TYPE "UDT_ModuleState"
TITLE = UDT_ModuleState
VERSION : 0.1
//User-defined structure of module states.
   STRUCT
      Configured { ExternalAccessible := 'False'; ExternalVisible := 'False'; ExternalWritable := 'False'} : Bool;   // Module configured
      Exist { ExternalAccessible := 'False'; ExternalVisible := 'False'; ExternalWritable := 'False'} : Bool;   // Module exist
      Error { ExternalAccessible := 'False'; ExternalVisible := 'False'; ExternalWritable := 'False'} : Bool;   // Module has error
   END_STRUCT;

END_TYPE

TYPE "UDT_DeviceState"
TITLE = UDT_DeviceState
VERSION : 0.1
//User-defined structure of device states.
   STRUCT
      Configure { ExternalAccessible := 'False'; ExternalVisible := 'False'; ExternalWritable := 'False'} : Bool;   // Device configured in TIA Portal hardware
      Exist { ExternalAccessible := 'False'; ExternalVisible := 'False'; ExternalWritable := 'False'} : Bool;   // Device physically connected
      Error { ExternalAccessible := 'False'; ExternalVisible := 'False'; ExternalWritable := 'False'} : Bool;   // Device has an error
      ProfinetNumber : UInt;   // Profinet slave number
      HW_ID : UInt;   // Device's HW_ID
      PNDeviceName : String;   // Device's project name
   END_STRUCT;

END_TYPE

TYPE "UDT_ProfinetDevice"
TITLE = UDT_ProfinetDevice
VERSION : 0.1
//User-defined structure of profinet device state.
   STRUCT
      DeviceState : "UDT_DeviceState";   // Device state
      Module { S7_SetPoint := 'False'} : Array[0..31] of "UDT_ModuleState";   // Modules
   END_STRUCT;

END_TYPE

TYPE "UDT_CommonStatus"
TITLE = UDT_CommonStatus
VERSION : 0.1
//User-defined structure of common statuses.
   STRUCT
      SafetyStop { ExternalAccessible := 'False'; ExternalVisible := 'False'; ExternalWritable := 'False'} : Bool;   // Emergancy stop
      Error { ExternalAccessible := 'False'; ExternalVisible := 'False'; ExternalWritable := 'False'} : Bool;   // An error is active
      Warning { ExternalAccessible := 'False'; ExternalVisible := 'False'; ExternalWritable := 'False'} : Bool;   // A warning is active
      ManualRun { ExternalAccessible := 'False'; ExternalVisible := 'False'; ExternalWritable := 'False'} : Bool;   // Running in manual mode
      Manual { ExternalAccessible := 'False'; ExternalVisible := 'False'; ExternalWritable := 'False'} : Bool;   // In manual mode
      Halted { ExternalAccessible := 'False'; ExternalVisible := 'False'; ExternalWritable := 'False'} : Bool;   // Halted
      Dieback { ExternalAccessible := 'False'; ExternalVisible := 'False'; ExternalWritable := 'False'} : Bool;   // In dieback
      Stopped { ExternalAccessible := 'False'; ExternalVisible := 'False'; ExternalWritable := 'False'} : Bool;   // Stopped
      Running { ExternalAccessible := 'False'; ExternalVisible := 'False'; ExternalWritable := 'False'} : Bool;   // Running
      EnergySave { ExternalAccessible := 'False'; ExternalVisible := 'False'; ExternalWritable := 'False'} : Bool;   // In energy saving mode
      AutoON { ExternalAccessible := 'False'; ExternalVisible := 'False'; ExternalWritable := 'False'} : Bool;   // Automatic started
   END_STRUCT;

END_TYPE

TYPE "UDT_ProfinetNetwork"
TITLE = UDT_ProfinetNetwork
VERSION : 0.1
//User-defined structure of profinet network state.
   STRUCT
      DeviceStatus : Array[0..512] of "UDT_ProfinetDevice";   // Profinet device status
   END_STRUCT;

END_TYPE

TYPE "UDT_GINWES"
VERSION : 0.1
   STRUCT
      Barcode : String[40];
   END_STRUCT;

END_TYPE

TYPE "UDT_GINWCS"
VERSION : 0.1
   STRUCT
      ActionTaken : String;   // Location code value that describes the actual disposition of the package
      Destination1 : String[20];   // Location code value that describes where the package should go (Diverter Number)
      Destination2 : String[20];   // Location code value that describes where the package should go (Diverter Number)
      Destination3 : String[20];   // Location code value that describes where the package should go (Diverter Number)
      Destination4 : String[20];   // Location code value that describes where the package should go (Diverter Number)
      Destination5 : String[20];   // Location code value that describes where the package should go (Diverter Number)
      ReasonCode : String[2];   // Management Code value that describes the result of attempting to route the package to the Destination
      Barcode1 : String;   // Barcode identifier code
      Barcode2 : String;
      Barcode3 : String;
      Barcode4 : String;
   END_STRUCT;

END_TYPE

TYPE "UDT_GINDHL"
VERSION : 0.1
   STRUCT
      ObjectID : String[10];   // Object ID
      VID : String[16];   // Virtual Item Identifier (VID)
      PieceID : String[40];   // Piece ID barcodes
      SortStrategy : String[1];   // Sort Strategy 1 - Highest priority available , 2 - Nearest
      ParcelReject { ExternalAccessible := 'False'; ExternalVisible := 'False'; ExternalWritable := 'False'} : Bool;   // True - Parcel reject
      Destination : Array[1..6] of Struct   // Destination
         ID : UInt;   // ID
         SortCommandActive { ExternalAccessible := 'False'; ExternalVisible := 'False'; ExternalWritable := 'False'} : Bool;   // Sort command
         ParcelSorted { ExternalAccessible := 'False'; ExternalVisible := 'False'; ExternalWritable := 'False'} : Bool;   // Parcel sorted
         Rejected { ExternalAccessible := 'False'; ExternalVisible := 'False'; ExternalWritable := 'False'} : Bool;   // Parcel rejected
         Reason : Int;   // Reason
      END_STRUCT;
      ParcelLocation : Struct   // Parcel Location
         Current : UInt;   // Current
         Last : UInt;   // Last
         Sort : UInt;   // Sort
      END_STRUCT;
      MFCMessage : Struct   // MFC Sort messages
         Sent : Struct   // Messages sent from the PLC to the MFC system
            SortResult { ExternalAccessible := 'False'; ExternalVisible := 'False'; ExternalWritable := 'False'} : Bool;   // Message Sort Result
            VIDResponse { ExternalAccessible := 'False'; ExternalVisible := 'False'; ExternalWritable := 'False'} : Bool;   // Message VID Response
            ScanReset { ExternalAccessible := 'False'; ExternalVisible := 'False'; ExternalWritable := 'False'} : Bool;   // Message Scan Reset
            XrayResult { ExternalAccessible := 'False'; ExternalVisible := 'False'; ExternalWritable := 'False'} : Bool;   // Message Xray result
            ParcelRegInfo { ExternalAccessible := 'False'; ExternalVisible := 'False'; ExternalWritable := 'False'} : Bool;   // Message Xray registration info
         END_STRUCT;
         Received : Struct   // Messages received from the MFC system to the PLC
            RejectParcel { ExternalAccessible := 'False'; ExternalVisible := 'False'; ExternalWritable := 'False'} : Bool;   // Message Reject Parcel
            Destination { ExternalAccessible := 'False'; ExternalVisible := 'False'; ExternalWritable := 'False'} : Bool;   // Message Destination
            DestinationResent { ExternalAccessible := 'False'; ExternalVisible := 'False'; ExternalWritable := 'False'} : Bool;   // Message Destination Resent
            TemporaryParcelIdentifier { ExternalAccessible := 'False'; ExternalVisible := 'False'; ExternalWritable := 'False'} : Bool;   // Message Temporary Parcel Identifier
            XrayRegistrationInfo { ExternalAccessible := 'False'; ExternalVisible := 'False'; ExternalWritable := 'False'} : Bool;
         END_STRUCT;
      END_STRUCT;
      Xray : Struct   // Xray data structure
         RoutingCode : String[2];   // Routing code
         Group : String[1];   // The group field is used to identify the group of the operator decisions came from in a
         Level : String[1];   // Level field is used to identify which level the operator decision came from in a
         Result : String[1];   // Results can be indicated with the following:A = Accept, R = Reject, U = Unavailable (Timeout), Z = High Threat
         BagIDMessage : Struct   // Message from PLC to Xray
            MessagePrepared { ExternalAccessible := 'False'; ExternalVisible := 'False'; ExternalWritable := 'False'} : Bool;   // The message is prepared and ready to send
            WrongMessageStructure { ExternalAccessible := 'False'; ExternalVisible := 'False'; ExternalWritable := 'False'} : Bool;   // The message has wrong structure
            Sent { ExternalAccessible := 'False'; ExternalVisible := 'False'; ExternalWritable := 'False'} : Bool;   // The message sent by PLC to Xray
            SentTime : String;   // Time when message sent by PLC to Xray
            NotSent { ExternalAccessible := 'False'; ExternalVisible := 'False'; ExternalWritable := 'False'} : Bool;   // The message was not sent from the PLC
            Received { ExternalAccessible := 'False'; ExternalVisible := 'False'; ExternalWritable := 'False'} : Bool;   // The message received by Xray
            TimeReceived : String;   // Time when message received by Xray
            NotReceived { ExternalAccessible := 'False'; ExternalVisible := 'False'; ExternalWritable := 'False'} : Bool;   // The message did not reach Xray
         END_STRUCT;
         DecisionMessage : Struct   // Message from Xray to PLC
            Received { ExternalAccessible := 'False'; ExternalVisible := 'False'; ExternalWritable := 'False'} : Bool;   // The message received by PLC
            ReceivedTime : String;   // The message received by PLC
            NotReceivedOnTime { ExternalAccessible := 'False'; ExternalVisible := 'False'; ExternalWritable := 'False'} : Bool;   // The message did not reach PLC
         END_STRUCT;
      END_STRUCT;
   END_STRUCT;

END_TYPE

TYPE "UDT_GINUPS"
VERSION : 0.1
   STRUCT
      TRKNUM : String[18];   // Tracking number
      PKGUID : String[32];   // Package ID
      MSGID : String[32];   // Message ID
      Length : Int;   // Camera Length in mm
      Width : Int;   // Camera Width in mm
      Height : Int;   // Camera Height in mm
      Weight : DInt;   // Weight in g
      IDCreated { ExternalAccessible := 'False'; ExternalVisible := 'False'; ExternalWritable := 'False'} : Bool;   // Byte 1, Bit 0 - PLCID created or TrayID Read
      DimDataRcv { ExternalAccessible := 'False'; ExternalVisible := 'False'; ExternalWritable := 'False'} : Bool;   // Byte 1, Bit 1 - Package Dimensional Data Received via Camera Scan Data Message
      PkgWrongInduct { ExternalAccessible := 'False'; ExternalVisible := 'False'; ExternalWritable := 'False'} : Bool;   // Byte 1, Bit 2 - Package Did NOT Induct Properly (Non-Tray Systems)
      IDCalcFromCamID { ExternalAccessible := 'False'; ExternalVisible := 'False'; ExternalWritable := 'False'} : Bool;   // Byte 2, Bit 0 - PLCID/TrayID Calculated From CamID
      UnknownParcelID { ExternalAccessible := 'False'; ExternalVisible := 'False'; ExternalWritable := 'False'} : Bool;   // Byte 2, Bit 4 - Unknown Parcel ID
      UndefinedProblem { ExternalAccessible := 'False'; ExternalVisible := 'False'; ExternalWritable := 'False'} : Bool;   // Byte 2, Bit 5 - Un-Defined Problem
      UnrecognizedCmd { ExternalAccessible := 'False'; ExternalVisible := 'False'; ExternalWritable := 'False'} : Bool;   // Byte 2, Bit 6 - Un-recognized command
      SorterInMainteneceMode { ExternalAccessible := 'False'; ExternalVisible := 'False'; ExternalWritable := 'False'} : Bool;   // Byte 2, Bit 7 - Sorter in Maintenance/Commissioning Mode
      DestUserSusp { ExternalAccessible := 'False'; ExternalVisible := 'False'; ExternalWritable := 'False'} : Bool;   // Byte 3, Bit 3 - Destination User Suspended
      SorterNotSynch { ExternalAccessible := 'False'; ExternalVisible := 'False'; ExternalWritable := 'False'} : Bool;   // Byte 3, Bit 6 - Sorter NOT Synchronized (Tilt Tray Systems)
      PkgDetAtVerCheckPoint { ExternalAccessible := 'False'; ExternalVisible := 'False'; ExternalWritable := 'False'} : Bool;   // Byte 4, Bit 0 - Package Detected at Verification Check Point
      ChuteFullAftrAlterDest { ExternalAccessible := 'False'; ExternalVisible := 'False'; ExternalWritable := 'False'} : Bool;   // Byte 4, Bit 7 - Preferred chute full after passed alternate destination
      ChuteNotAvailAfterAlterDest { ExternalAccessible := 'False'; ExternalVisible := 'False'; ExternalWritable := 'False'} : Bool;   // Byte 5, Bit 0 - Preferred chute not available after passed alternate destination
      PLCRedirected { ExternalAccessible := 'False'; ExternalVisible := 'False'; ExternalWritable := 'False'} : Bool;   // Byte 5, Bit 2 - PLC Redirected
      ThreatParcel { ExternalAccessible := 'False'; ExternalVisible := 'False'; ExternalWritable := 'False'} : Bool;   // Threat parcel
   END_STRUCT;

END_TYPE

TYPE "UDT_GINFedEx"
VERSION : 0.1
   STRUCT
      Timestamp : String[17];   // Local time timestamp
      TimeZoneDesignator : String[5];   // Time zone designator
      PackageEntrancePoint : String[14];   // Entrance point, where LLC starts tracking the parcel.
      PackageEntranceState : String[1];   // Entrance state
      PackageExitPoint : String[14];   // Exit point name, where LLC reports the last known tracking point.
      PackageExitState : String[1];   // Exit point state when LLC reports the last known tracking point.
      PalletType : String[2];   // Pallet code for different type of pallets on the market
      Mask : String[1];   // Flag to indicate that a pallet has been mask.
      CellNumber : String[4];   // Tray/Cell number (for loop sorters) or generated by LLC (on line sorters).
      CellsOccupied : String[1];   // Cells occupied by the piece for loop sorters.
      ImageID : String[6];   // Image ID number created by the ADC system.
      ScanUnitType : String[1];   // Scan unit type
      ADCSystemID : String[15];   // Number assigned by the ADC system
      PackageID : String[15];   // Number assigned by the LLC system
      LLCSystemID : String[15];
      HLCPackageID : String[10];   // Unique number for the specific package during it stays in HLC system.
      HLCResultCode : String[16];   // Result code based on processing of the scan event messages.
      ShipmentID : String[6];   // Consignment id of the parcel.
      WeightStatus : String[1];   // Status to indicate if the parcel/pallet has weight on the system.
      ActualDestination : String[6];   // Location code value that describes the actual disposition of the package.
      Destination1 : String[6];   // Location code value that describes where the package should go (Diverter Number).
      Destination2 : String[6];   // Location code value that describes where the package should go (Diverter Number).
      Destination3 : String[6];   // Location code value that describes where the package should go (Diverter Number).
      Destination4 : String[6];   // Location code value that describes where the package should go (Diverter Number).
      Destination5 : String[6];   // Location code value that describes where the package should go (Diverter Number).
      CutOffTimeDestination1 : String[5];   // Cut Off Time in Local Time.
      CutOffTimeDestination2 : String[5];   // Cut Off Time in Local Time.
      CutOffTimeDestination3 : String[5];   // Cut Off Time in Local Time.
      CutOffTimeDestination4 : String[5];   // Cut Off Time in Local Time.
      CutOffTimeDestination5 : String[5];   // Cut Off Time in Local Time.
      ReasonCode1 : String[8];   // Management Code value that describes the result of attempting to route the package to the Destination
      ReasonCode2 : String[8];   // Management Code value that describes the result of attempting to route the package to the Destination
      ReasonCode3 : String[8];   // Management Code value that describes the result of attempting to route the package to the Destination
      ReasonCode4 : String[8];   // Management Code value that describes the result of attempting to route the package to the Destination
      ReasonCode5 : String[8];   // Management Code value that describes the result of attempting to route the package to the Destination
      HLCDataText : String[20];   // Free text for future use.
      Customs : String[1];   // Need to be checked by customs
      DIMSystemID : String[15];   // Identifier of dimensioning system.
      DIMStatus : String[5];   // Basic diagnostic information from the dimensioning system at the moment of the measurement.
      PackageDimLength : String[6];   // Length dimension of package in resolution of dim system.
      PackageDimWidth : String[6];   // Width dimension of package in resolution of dim system.
      PackageDimHeight : String[6];   // Height dimension of package in resolution of dim system.
      DIMUOM : String[2];   // Unit of measure of the package dimensions.
      DimLFTstatusCode : String[8];   // Dimension LFT status code.
      DimConfidence : String[2];   // The level of assurance for the correct dimensions.
      DimensionSource : String[1];   // For combined camera/laser dim acquisition devices. It indicates type of capturing mode
      AlibiDims : String[25];   // Alibi for Dimensions
      SCLSystemID : String[15];   // Identifier of weight scale.
      SCLStatus : String[5];   // Basic diagnostic information from the weight scale system.
      SCLWT : String[6];   // Scale weight of package in resolution of scale system.
      SCLWTUOM : String[2];   // Unit of measurement for Weight
      SCLLFTStatusCode : String[2];   // Scale LFT status code.
      AlibiWeight : String[25];   // Alibi for Weight
      ReasonCode : String[1];   // This code should be used when the SI message has some defect.
      Stackable : String[1];   // If stackable recognition is enabled, Y or N
      Stickerstype : String[2];   // When optical recognition is used to sort
      FlyingDocument : String[1];   // Status to confirm if the document/flyer is prone to fly off the sorter.
      ModeofOperation : String[1];   // Camera Tunnel operational mode format:
      CameraHeadstatus : String[2];   // Diagnostic information on camera/laser heads performing barcode reads.
      PackageDataTruncated : String[1];   // Y = Full length of barcode data exceeds 9999 bytes, data truncated
      TotalBarcodeDataLength : String[4];   // Length of all barcode data that was sent in bytes;
      Barcode1Identification : String[3];   // Barcode identifier code.
      Barcode1status : String[2];   // Barcode confidence factor
      Barcode1datalength : String[4];   // String length of barcode data in bytes; inclusive of this field. Use 0054 as a fixed value
      Barcode1data : String[50];   // Highest priority barcode
      Barcode2Identification : String[3];   // Barcode identifier code.
      Barcode2status : String[2];   // Barcode confidence factor
      Barcode2datalength : String[4];   // String length of barcode data in bytes; inclusive of this field. Use 0054 as a fixed value
      Barcode2data : String[50];   // Highest priority barcode
      Barcode3Identification : String[3];   // Barcode identifier code.
      Barcode3status : String[2];   // Barcode confidence factor
      Barcode3datalength : String[4];   // String length of barcode data in bytes; inclusive of this field. Use 0054 as a fixed value
      Barcode3data : String[50];   // Highest priority barcode
      BarcodeIdentification : String[3];   // Barcode identifier code.
      Barcodestatus : String[2];   // Barcode confidence factor
      Barcodedatalength : String[4];   // String length of barcode data in bytes
      Barcodedata : String[50];   // Sortation barcode
      CustomerID : DInt;   // 6 digits SequentialID (NNNNNN)
      AreaNumber : String[2];   // Package Sequence ID "Area Number"
      PurgeEnabled { ExternalAccessible := 'False'; ExternalVisible := 'False'; ExternalWritable := 'False'} : Bool;   // Purge enabled for parcel: destination overwritten with Purge destination
   END_STRUCT;

END_TYPE

TYPE "UDT_GINStandard"
VERSION : 0.1
   STRUCT
      Destination : Array[0..20] of DInt;   // Destination
      Identification : Struct   // Barcode identification
         GoodRead { ExternalAccessible := 'False'; ExternalVisible := 'False'; ExternalWritable := 'False'} : Bool;   // Barcode read was succesful
         NoRead { ExternalAccessible := 'False'; ExternalVisible := 'False'; ExternalWritable := 'False'} : Bool;   // Barcode read was unsuccesful
         MultiRead { ExternalAccessible := 'False'; ExternalVisible := 'False'; ExternalWritable := 'False'} : Bool;   // Multiple Barcodes were detected
         Barcode : Array[0..10] of Char;   // Barcode values
      END_STRUCT;
      GinAssigned { ExternalAccessible := 'False'; ExternalVisible := 'False'; ExternalWritable := 'False'} : Bool;   // GIN is assigned to package
      Lost { ExternalAccessible := 'False'; ExternalVisible := 'False'; ExternalWritable := 'False'} : Bool;   // Lost in tracking
      Length : Int;   // Length in mm
      Width : Int;   // Width in mm
      Height : Int;   // Height in mm
      Weight : DInt;   // Weight in g
      PkgTooLong { ExternalAccessible := 'False'; ExternalVisible := 'False'; ExternalWritable := 'False'} : Bool;   // Package is too long
      PkgTooSmall { ExternalAccessible := 'False'; ExternalVisible := 'False'; ExternalWritable := 'False'} : Bool;   // Package is too small
      PkgTooHigh { ExternalAccessible := 'False'; ExternalVisible := 'False'; ExternalWritable := 'False'} : Bool;   // Package is too high
      PkgOverWeight { ExternalAccessible := 'False'; ExternalVisible := 'False'; ExternalWritable := 'False'} : Bool;   // Package is over weight
      TrailingGap : Int;   // Trailing gap size in cm between the package
      LeadingGap : Int;   // Leading gap size in cm between the package
      NrOfRecirculations : Int;   // Number of recirculations
      DestReqSend { ExternalAccessible := 'False'; ExternalVisible := 'False'; ExternalWritable := 'False'} : Bool;   // Destination request sent to high level
      DestRcv { ExternalAccessible := 'False'; ExternalVisible := 'False'; ExternalWritable := 'False'} : Bool;   // Destination received from high level
      SortStatus : Struct   // Sort status of the package
         DivertDestination : Int;   // Destination to which the package is diverted
         GoodDivert { ExternalAccessible := 'False'; ExternalVisible := 'False'; ExternalWritable := 'False'} : Bool;   // Package diverted
         FailedDivert { ExternalAccessible := 'False'; ExternalVisible := 'False'; ExternalWritable := 'False'} : Bool;   // Package failed to divert
         NoDivert : Bool := TRUE;   // Divert is not activated
         NoDivertCause : Struct   // Cause for no divert
            ChuteJam { ExternalAccessible := 'False'; ExternalVisible := 'False'; ExternalWritable := 'False'} : Bool;   // Chute is jammed
            ChuteFull { ExternalAccessible := 'False'; ExternalVisible := 'False'; ExternalWritable := 'False'} : Bool;   // Chute is full
            NoRTR { ExternalAccessible := 'False'; ExternalVisible := 'False'; ExternalWritable := 'False'} : Bool;   // Downstream conveyor is not ready to receive
            DestDisabled { ExternalAccessible := 'False'; ExternalVisible := 'False'; ExternalWritable := 'False'} : Bool;   // Destination is disabled
            TrayDisabled { ExternalAccessible := 'False'; ExternalVisible := 'False'; ExternalWritable := 'False'} : Bool;   // Tray is disabled
            SorterNotAtSpeed { ExternalAccessible := 'False'; ExternalVisible := 'False'; ExternalWritable := 'False'} : Bool;   // Sorter is not at speed
            LeadingGapError { ExternalAccessible := 'False'; ExternalVisible := 'False'; ExternalWritable := 'False'} : Bool;   // Gap size with downstream parcel is not enough
            TrailingGapError { ExternalAccessible := 'False'; ExternalVisible := 'False'; ExternalWritable := 'False'} : Bool;   // Gap size with upstream parcel is not enough
            PkgTooHigh { ExternalAccessible := 'False'; ExternalVisible := 'False'; ExternalWritable := 'False'} : Bool;   // Package is too high to divert
            PkgTooLong { ExternalAccessible := 'False'; ExternalVisible := 'False'; ExternalWritable := 'False'} : Bool;   // Package is too long to divert
            DestNotReachable { ExternalAccessible := 'False'; ExternalVisible := 'False'; ExternalWritable := 'False'} : Bool;   // Sort destionation is not reachable
            InvalidDest { ExternalAccessible := 'False'; ExternalVisible := 'False'; ExternalWritable := 'False'} : Bool;   // Sort destination is invalid
            DestTooLate { ExternalAccessible := 'False'; ExternalVisible := 'False'; ExternalWritable := 'False'} : Bool;   // Destination too late
            NoDestRcv { ExternalAccessible := 'False'; ExternalVisible := 'False'; ExternalWritable := 'False'} : Bool;   // Destination not received from high level
         END_STRUCT;
      END_STRUCT;
   END_STRUCT;

END_TYPE

TYPE "UDT_EventStatistic"
TITLE = UDT_EventStatistic
VERSION : 0.1
//User-defined structure of event statistic data.
   STRUCT
      NumberOfTimes : DInt;   // Number of times the event occurred since last reset
      LastEventSeconds : DInt;   // Number of seconds of the current or last event
      TotalEventSeconds : DInt;   // Total number of seconds the event occurred since last reset
   END_STRUCT;

END_TYPE

FUNCTION "FC_GetNrOfArrayEl" : Int
TITLE = FC_GetNrOfArrayEl
{ S7_Optimized_Access := 'TRUE' }
AUTHOR : MHSE
FAMILY : GeneralSystemFunctions
VERSION : 3.0
// ATTRIBUTES
// AUTO_NUMBER = True
// BLOCK_NUMBER = 19
// END_ATTRIBUTES
//Function to get the number of array elements.
   VAR_INPUT
      iv_Array : Variant;   // Input array
   END_VAR

   VAR_TEMP
      ti_NrOfArrayEl : Int;   // Number of array elements
   END_VAR


BEGIN
	(*
	----------------------------------------------------------------------------------------

	Version history:
	Date        | Version   | Author        | Remark
	----------------------------------------------------------------------------------------
	24/05/2019  | 0.1       | L.Klar        | first release MHS TIA 15.1
	24/07/2019  | 2.0       | L.Klar        | 2.0 MHS library release TIA 15.1
	27/08/2019  | 2.1       | K.Pokorski    | Comments adjusted
	12/11/2019  | 3.0       | P.Majka       | 3.0 MHS library release TIA 15.1
	21/02/2023  | 4.0       | F.Baten       | 4.0 Release TIA 17.5
	*)

	REGION 1 – Number of an array elements

	    IF IS_ARRAY(#iv_Array)                                                  // Input variable is an array
	    THEN

	        #ti_NrOfArrayEl := UDINT_TO_INT(CountOfElements(#iv_Array));

	        // Reset array length if the input variable isn't an array
	    ELSE

	        #ti_NrOfArrayEl := 0;

	    END_IF;

	END_REGION

	REGION 2 – Return output

	    #FC_GetNrOfArrayEl := #ti_NrOfArrayEl;

	END_REGION

END_FUNCTION

TYPE "UDT_AixMotorStatus"
VERSION : 0.1
   STRUCT
      Overheat { ExternalAccessible := 'False'; ExternalVisible := 'False'; ExternalWritable := 'False'} : Bool;   // Motor temperature has exceeded 105 degrees Celsius
      MaxTorque { ExternalAccessible := 'False'; ExternalVisible := 'False'; ExternalWritable := 'False'} : Bool;   // Motor at maximum torque output
      ShortCircuit { ExternalAccessible := 'False'; ExternalVisible := 'False'; ExternalWritable := 'False'} : Bool;   // Motor short circuit
      MotorNotConnected { ExternalAccessible := 'False'; ExternalVisible := 'False'; ExternalWritable := 'False'} : Bool;   // Motor is not connected
      Overload { ExternalAccessible := 'False'; ExternalVisible := 'False'; ExternalWritable := 'False'} : Bool;   // Motor overloaded after more than 20 seconds in Stalled
      Stalled { ExternalAccessible := 'False'; ExternalVisible := 'False'; ExternalWritable := 'False'} : Bool;   // Motor stalled and speed is less than 10% of the set speed
      BadHall { ExternalAccessible := 'False'; ExternalVisible := 'False'; ExternalWritable := 'False'} : Bool;   // Motor Hall Effect Sensor error active
      MotorNotUsed { ExternalAccessible := 'False'; ExternalVisible := 'False'; ExternalWritable := 'False'} : Bool;   // Motor is not used
      MotorStatus1 { ExternalAccessible := 'False'; ExternalVisible := 'False'; ExternalWritable := 'False'} : Bool;   // Motor running and direction status
      MotorStatus2 { ExternalAccessible := 'False'; ExternalVisible := 'False'; ExternalWritable := 'False'} : Bool;   // Motor running and direction status
      MotorPortinDOmode { ExternalAccessible := 'False'; ExternalVisible := 'False'; ExternalWritable := 'False'} : Bool;   // Motor port is in digital output mode .
      Bit03 { ExternalAccessible := 'False'; ExternalVisible := 'False'; ExternalWritable := 'False'} : Bool;   // Reserved
      Bit04 { ExternalAccessible := 'False'; ExternalVisible := 'False'; ExternalWritable := 'False'} : Bool;   // Reserved
      BoardOverheat { ExternalAccessible := 'False'; ExternalVisible := 'False'; ExternalWritable := 'False'} : Bool;   // Reserved
      OverVoltage { ExternalAccessible := 'False'; ExternalVisible := 'False'; ExternalWritable := 'False'} : Bool;   // Supply voltage + motor back EMF exceeded 30 volts
      LowVoltage { ExternalAccessible := 'False'; ExternalVisible := 'False'; ExternalWritable := 'False'} : Bool;   // Module power supply is less than 18 Volts
      MotorStatus : DWord;
   END_STRUCT;

END_TYPE

TYPE "UDT_EquipmentControl"
TITLE = UDT_EquipmentControl
VERSION : 0.1
//User-defined structure of equipment control commands.
   STRUCT
      Command : Struct   // Control command
         Start { ExternalAccessible := 'False'; ExternalVisible := 'False'; ExternalWritable := 'False'} : Bool;   // Start conveyor
         Stop { ExternalAccessible := 'False'; ExternalVisible := 'False'; ExternalWritable := 'False'} : Bool;   // Stop conveyor
         Reset { ExternalAccessible := 'False'; ExternalVisible := 'False'; ExternalWritable := 'False'} : Bool;   // Faults reset
         ResetData { ExternalAccessible := 'False'; ExternalVisible := 'False'; ExternalWritable := 'False'} : Bool;   // Statistics reset
         ManualMode { ExternalAccessible := 'False'; ExternalVisible := 'False'; ExternalWritable := 'False'} : Bool;   // Manual mode required
         DisableManualMode { ExternalAccessible := 'False'; ExternalVisible := 'False'; ExternalWritable := 'False'} : Bool;   // Disable manual mode
         AutomaticOn { ExternalAccessible := 'False'; ExternalVisible := 'False'; ExternalWritable := 'False'} : Bool;   // System is started in automatic mode
         StopRequest { ExternalAccessible := 'False'; ExternalVisible := 'False'; ExternalWritable := 'False'} : Bool;
      END_STRUCT;
      Report { S7_SetPoint := 'False'} : "UDT_CommonStatus";   // Conveyors state
      Request : Struct   // Request from equipment
         RestartRequired { ExternalAccessible := 'False'; ExternalVisible := 'False'; ExternalWritable := 'False'} : Bool;   // Restart required from system control
         SignalingRequest { ExternalAccessible := 'False'; ExternalVisible := 'False'; ExternalWritable := 'False'} : Bool;   // Beeper required
         InhibitStop { ExternalAccessible := 'False'; ExternalVisible := 'False'; ExternalWritable := 'False'} : Bool;
      END_STRUCT;
   END_STRUCT;

END_TYPE

DATA_BLOCK "DB_ProfinetDiagnostic"
TITLE = DB_ProfinetDiagnostic
{ S7_Optimized_Access := 'TRUE' }
AUTHOR : MHSE
FAMILY : GeneralSystemFunctions
VERSION : 3.0
NON_RETAIN
//Data block to store profinet network diagnostic data.
   VAR
      ProfinetNetworks { ExternalAccessible := 'False'; ExternalVisible := 'False'; ExternalWritable := 'False'; S7_SetPoint := 'False'} : Array[1..10] of "UDT_ProfinetNetwork";
   END_VAR


BEGIN

END_DATA_BLOCK

TYPE "UDT_GIN"
VERSION : 0.1
   STRUCT
      General { S7_SetPoint := 'False'} : "UDT_GINStandard";
      FedEx { S7_SetPoint := 'False'} : "UDT_GINFedEx";
      UPS { S7_SetPoint := 'False'} : "UDT_GINUPS";
      DHL { S7_SetPoint := 'False'} : "UDT_GINDHL";
      WCS { S7_SetPoint := 'False'} : "UDT_GINWCS";
      WES { S7_SetPoint := 'False'} : "UDT_GINWES";
   END_STRUCT;

END_TYPE

DATA_BLOCK "DB_Memory"
TITLE = DB_Memory
{ S7_Optimized_Access := 'TRUE' }
AUTHOR : MHSE
VERSION : 3.0
NON_RETAIN
   VAR
      ClockByte { ExternalAccessible := 'False'; ExternalVisible := 'False'; ExternalWritable := 'False'} : Byte;   // System clock byte
      Clock_10Hz { ExternalAccessible := 'False'; ExternalVisible := 'False'; ExternalWritable := 'False'} : Bool;   // 10 Hz system clock bit
      Clock_5Hz { ExternalAccessible := 'False'; ExternalVisible := 'False'; ExternalWritable := 'False'} : Bool;   // 5 Hz system clock bit
      "Clock_2.5Hz" { ExternalAccessible := 'False'; ExternalVisible := 'False'; ExternalWritable := 'False'} : Bool;   // 2.5 Hz system clock bit
      Clock_2Hz { ExternalAccessible := 'False'; ExternalVisible := 'False'; ExternalWritable := 'False'} : Bool;   // 2 Hz system clock bit
      "Clock_1.25Hz" { ExternalAccessible := 'False'; ExternalVisible := 'False'; ExternalWritable := 'False'} : Bool;   // 1.25 Hz system clock bit
      Clock_1Hz { ExternalAccessible := 'False'; ExternalVisible := 'False'; ExternalWritable := 'False'} : Bool;   // 1 Hz system clock bit
      "Clock_0.625Hz" { ExternalAccessible := 'False'; ExternalVisible := 'False'; ExternalWritable := 'False'} : Bool;   // 0.625 Hz system clock bit
      "Clock_0.5Hz" { ExternalAccessible := 'False'; ExternalVisible := 'False'; ExternalWritable := 'False'} : Bool;   // 0.5 Hz system clock bit
      SystemByte { ExternalAccessible := 'False'; ExternalVisible := 'False'; ExternalWritable := 'False'} : Byte;   // System byte
      OSClockByte { ExternalAccessible := 'False'; ExternalVisible := 'False'; ExternalWritable := 'False'} : Byte;   // One shot of clock pulse
      "OS_0.1sec" { ExternalAccessible := 'False'; ExternalVisible := 'False'; ExternalWritable := 'False'} : Bool;   // One shot every 0.1 sec
      "OS_0.2sec" { ExternalAccessible := 'False'; ExternalVisible := 'False'; ExternalWritable := 'False'} : Bool;   // One shot every 0.2 sec
      "OS_0.4sec" { ExternalAccessible := 'False'; ExternalVisible := 'False'; ExternalWritable := 'False'} : Bool;   // One shot every 0.4 sec
      "OS_0.5sec" { ExternalAccessible := 'False'; ExternalVisible := 'False'; ExternalWritable := 'False'} : Bool;   // One shot every 0.5 sec
      "OS_0.8sec" { ExternalAccessible := 'False'; ExternalVisible := 'False'; ExternalWritable := 'False'} : Bool;   // One shot every 0.8 sec
      OS_1sec { ExternalAccessible := 'False'; ExternalVisible := 'False'; ExternalWritable := 'False'} : Bool;   // One shot every 1 sec
      "OS_1.6sec" { ExternalAccessible := 'False'; ExternalVisible := 'False'; ExternalWritable := 'False'} : Bool;   // One shot every 1.6 sec
      OS_2sec { ExternalAccessible := 'False'; ExternalVisible := 'False'; ExternalWritable := 'False'} : Bool;   // One shot every 2 sec
      PrevCycleTime { ExternalAccessible := 'False'; ExternalVisible := 'False'; ExternalWritable := 'False'} : LReal;   // Previous PLC cycle Time
      RuntimeMem { ExternalAccessible := 'False'; ExternalVisible := 'False'; ExternalWritable := 'False'} : LReal;   // Runtime memory
      FirstScan { ExternalAccessible := 'False'; ExternalVisible := 'False'; ExternalWritable := 'False'} : Bool;   // First scan bit
      DiagStatusUpdate { ExternalAccessible := 'False'; ExternalVisible := 'False'; ExternalWritable := 'False'} : Bool;   // Diagnostic status update
      AlwaysTrue { ExternalAccessible := 'False'; ExternalVisible := 'False'; ExternalWritable := 'False'} : Bool;   // Always True bit
      AlwaysFalse { ExternalAccessible := 'False'; ExternalVisible := 'False'; ExternalWritable := 'False'} : Bool;   // Always False bit
      CommissioningFalse { ExternalAccessible := 'False'; ExternalVisible := 'False'; ExternalWritable := 'False'} : Bool;   // Commissioning always false
      CommissioningTrue { ExternalAccessible := 'False'; ExternalVisible := 'False'; ExternalWritable := 'False'} : Bool;   // Commissioning always true
      ReconnectCommand { ExternalAccessible := 'False'; ExternalVisible := 'False'; ExternalWritable := 'False'} : Bool;   // Reconnect command
      ScanMainRack { ExternalAccessible := 'False'; ExternalVisible := 'False'; ExternalWritable := 'False'} : Bool;   // Trigger to check main rack confiuration
      ScanProfinet { ExternalAccessible := 'False'; ExternalVisible := 'False'; ExternalWritable := 'False'} : Bool;   // Scan profinet bit
      Simulation { ExternalAccessible := 'False'; ExternalVisible := 'False'; ExternalWritable := 'False'} : Bool;   // Simulation
      PN1OK { ExternalAccessible := 'False'; ExternalVisible := 'False'; ExternalWritable := 'False'} : Bool;   // Profinet ok
      "Local~PROFINET_IO-System" { ExternalAccessible := 'False'; ExternalVisible := 'False'; ExternalWritable := 'False'} : HW_ANY;   // HW Intentifier of PN-IO System
      "Local~PROFINET_IO-System_1" { ExternalAccessible := 'False'; ExternalVisible := 'False'; ExternalWritable := 'False'} : HW_ANY;   // HW Intentifier of PN-IOSystem 1
      "Local~PROFINET_IO-System_2" { ExternalAccessible := 'False'; ExternalVisible := 'False'; ExternalWritable := 'False'} : HW_ANY;   // HW Intentifier of PN-IOSystem 2
      "Local~PROFINET_IO-System_3" { ExternalAccessible := 'False'; ExternalVisible := 'False'; ExternalWritable := 'False'} : HW_ANY;   // HW Intentifier of PN-IOSystem 3
      "Local~PROFINET_IO-System_4" { ExternalAccessible := 'False'; ExternalVisible := 'False'; ExternalWritable := 'False'} : HW_ANY;   // HW Intentifier of PN-IOSystem 4
      "Local~PROFINET_IO-System_5" { ExternalAccessible := 'False'; ExternalVisible := 'False'; ExternalWritable := 'False'} : HW_ANY;   // HW Intentifier of PN-IOSystem 5
      "Local~PROFINET_IO-System_6" { ExternalAccessible := 'False'; ExternalVisible := 'False'; ExternalWritable := 'False'} : HW_ANY;   // HW Intentifier of PN-IOSystem 6
      "Local~PROFINET_IO-System_7" { ExternalAccessible := 'False'; ExternalVisible := 'False'; ExternalWritable := 'False'} : HW_ANY;   // HW Intentifier of PN-IOSystem 7
      "Local~PROFINET_IO-System_8" { ExternalAccessible := 'False'; ExternalVisible := 'False'; ExternalWritable := 'False'} : HW_ANY;   // HW Intentifier of PN-IOSystem 8
      "Local~PROFINET_IO-System_9" { ExternalAccessible := 'False'; ExternalVisible := 'False'; ExternalWritable := 'False'} : HW_ANY;   // HW Intentifier of PN-IOSystem 9
   END_VAR


BEGIN

END_DATA_BLOCK

TYPE "UDT_PNDevice"
VERSION : 0.1
   STRUCT
      PNNetworknumber : Int := 1;   // Number of the profinet network where device exist
      PNDeviceNumber : Int := 0;   // Profinet number of the device
      PNDeviceFound { ExternalAccessible := 'False'; ExternalVisible := 'False'; ExternalWritable := 'False'} : Bool;   // Device found in Profinet structure
   END_STRUCT;

END_TYPE

TYPE "UDT_VfdSinaParameterUser"
TITLE = UDT_VFD_SinaParameterUser
VERSION : 0.1
//User-defined structure of Siemens parameter.
   STRUCT
      siParaNo : UInt;   // Number of parameter (Number 1..65535)
      siIndex : Int;   // Subindex (Number 1..65535)
      srValue : Real;   // Value of parameter
      sdValue : DInt;   // Value of parameter
      syFormat : Byte := BYTE#16#00;   // Format of value (Format 0x40..0x44)
      swErrorNo : Word := WORD#16#0000;   // Error number (see table below)
   END_STRUCT;

END_TYPE

TYPE "UDT_ConveyorCommonConfiguration"
VERSION : 0.1
   STRUCT
      Length : DInt;   // Conveyor length [mm]
      LengthCorrection : DInt;   // Length correction [mm]
   END_STRUCT;

END_TYPE

TYPE "UDT_InductParcelData"
VERSION : 0.1
   STRUCT
      GINNumber : Int;   // GIN number
      GapRequired : Int;   // Size of gap requested by induct
      WindowPosition : Int;   // Position of the window in the merge tracking
      WindowReserved { ExternalAccessible := 'False'; ExternalVisible := 'False'; ExternalWritable := 'False'} : Bool;   // The window is reserved for the induct
   END_STRUCT;

END_TYPE

FUNCTION_BLOCK "FB_OnOffDelayDistance"
TITLE = FB_TimerOnOffDelay
{ S7_Optimized_Access := 'TRUE' }
AUTHOR : MHSE
FAMILY : GeneralSystemFunctions
VERSION : 3.0
// ATTRIBUTES
// AUTO_NUMBER = True
// BLOCK_NUMBER = 18
// END_ATTRIBUTES
//Function block to generate on/off signal delay.
   VAR_INPUT
      idi_OnDelayDistance { ExternalAccessible := 'False'; ExternalVisible := 'False'; ExternalWritable := 'False'} : DInt;   // On delay distance [cm]
      idi_OffDelayDistance { ExternalAccessible := 'False'; ExternalVisible := 'False'; ExternalWritable := 'False'} : DInt;   // Off delay distance [cm]
      ii_Displacement { ExternalAccessible := 'False'; ExternalVisible := 'False'; ExternalWritable := 'False'} : Int;   // Actual displacement
      ix_SignalToDelay { ExternalAccessible := 'False'; ExternalVisible := 'False'; ExternalWritable := 'False'} : Bool;   // Input signal to be delayed
      ix_Enable { ExternalAccessible := 'False'; ExternalVisible := 'False'; ExternalWritable := 'False'} : Bool := TRUE;   // Measuring enable
   END_VAR

   VAR_OUTPUT
      qdi_ActualDelayDistance { ExternalAccessible := 'False'; ExternalVisible := 'False'; ExternalWritable := 'False'} : DInt;   // Actual delay distance [cm]
      qx_DelayedSignal { ExternalAccessible := 'False'; ExternalVisible := 'False'; ExternalWritable := 'False'} : Bool;   // Delayed signal output
   END_VAR

   VAR RETAIN
      sdi_ActualDelayDistance { ExternalAccessible := 'False'; ExternalVisible := 'False'; ExternalWritable := 'False'} : DInt;   // Actual delay distance [cm]
   END_VAR
   VAR
      s_R_TRIG_Signal {InstructionName := 'R_TRIG'; LibVersion := '1.0'; ExternalAccessible := 'False'; ExternalVisible := 'False'; ExternalWritable := 'False'; S7_SetPoint := 'False'} : R_TRIG;   // Siemens "R_Trig" - to prepare the rising edge trigger on "ix_SignalToDelay" signal
      s_F_TRIG_Signal {InstructionName := 'F_TRIG'; LibVersion := '1.0'; ExternalAccessible := 'False'; ExternalVisible := 'False'; ExternalWritable := 'False'; S7_SetPoint := 'False'} : F_TRIG;   // Siemens "F_Trig" - to prepare the falling edge trigger on "ix_SignalToDelay" signal
   END_VAR


BEGIN
	(*
	----------------------------------------------------------------------------------------

	Version history:
	Date        | Version   | Author        | Remark
	----------------------------------------------------------------------------------------
	26/04/2023  | 0.1       | F.Baten       | first release MHS TIA 15.1
	*)

	REGION Step 1 – Input signal edge detection

	    #s_R_TRIG_Signal(CLK := #ix_SignalToDelay);


	    #s_F_TRIG_Signal(CLK := #ix_SignalToDelay);

	END_REGION

	REGION Step 2 – Actual delay distance initialization

	    IF (#s_R_TRIG_Signal.Q OR #s_F_TRIG_Signal.Q)           // Input signal changed
	    THEN

	        #sdi_ActualDelayDistance := 0;

	    END_IF;

	END_REGION

	REGION Step 3 – On/Off delay distance calculation


	    IF (#ix_SignalToDelay                                       // Signal to be delayed is active
	        AND #ix_Enable)                                         // Measuring enabled
	    THEN

	        // Timer on
	        IF (#sdi_ActualDelayDistance >= #idi_OnDelayDistance)
	        THEN

	            #qx_DelayedSignal := TRUE;

	        ELSE

	            #sdi_ActualDelayDistance += ABS(#ii_Displacement);

	        END_IF;

	    END_IF;

	    // Timer off
	    IF (NOT #ix_SignalToDelay                                   // Signal to be delayed is not active
	        AND #ix_Enable)                                         // Measuring enabled
	    THEN

	        IF (#sdi_ActualDelayDistance >= #idi_OffDelayDistance)
	        THEN

	            #qx_DelayedSignal := FALSE;

	        ELSE

	            #sdi_ActualDelayDistance += ABS(#ii_Displacement);

	        END_IF;

	    END_IF;

	END_REGION

	REGION Step 4 – Actual time

	    #qdi_ActualDelayDistance := #sdi_ActualDelayDistance;

	END_REGION
END_FUNCTION_BLOCK

TYPE "UDT_PECDConfiguration"
VERSION : 0.1
   STRUCT
      Distance : DInt;   // Distance between photo eye and the end of conveyor [mm]
      OnDelayDistance : DInt;   // Photo eye distance on delay [cm]
      OffDelayDistance : DInt;   // Photo eye distance off delay [cm]
      JamDisplacementLimit : Int;   // Limit displacement with PEC blocked o detect jam [cm]
      ResetWithPECBlocked : Bool := TRUE;   // When 'True' Allow reset system after jam with PEC blocked
   END_STRUCT;

END_TYPE

TYPE "UDT_MotorData"
VERSION : 0.1
   STRUCT
      MainVoltage : Int;   // [Volt] Mains
      NominalVoltage : Int;   // [Volt] Motor nameplate for applicable connection
      NominalCurrent : Real;   // [Amps] Motor nameplate for applicable connection
      NominalPower : Real;   // [kW] Motor nameplate
      NominalSpeed : Int;   // [RPM] Motor nameplate
      NominalTorque : Real;   // [Nm] Motor nameplate
      CosPhi : Real;   // 0.0 - 0.99 Motor nameplate
      Connection : Int;   // 0=Start , 1=Delta
      BrakeConfig { ExternalAccessible := 'False'; ExternalVisible := 'False'; ExternalWritable := 'False'} : Bool;   // TRUE = Brake control from VFD. FALSE = No Brake
      EncoderConfig { ExternalAccessible := 'False'; ExternalVisible := 'False'; ExternalWritable := 'False'} : Bool;   // TRUE = Encoder connected at the VFD . FALSE = No encoder at the VFD
      EncoderResolution : Int;   // Pulses Per Rev
      ThermalConfig : Int;   // 0=No thermal control, 1= PTC1, 2=KTY84, 4= Bimetalic Switch
      NoMotorsParallel : Int;   // Number of motors in parallel
      VFDType : Int;   // Specific code 1= G120C, 5302= G120D 0,75kW, 5304= G120D 1,5kW, 5306= G120D 3kW, 5307= G120D 4kW, 5308= 5,5kW, 5309= G120D 7,5kW
      MinimumRamp : Int;   // Minimum applicable ramp in ms
      FAdress : Real;   // Safety adress from HW configuration
   END_STRUCT;

END_TYPE

TYPE "UDT_InductGapsize"
VERSION : 0.1
   STRUCT
      "Maximal length" : Int;   // Maximal length of parcel [cm]
      Gap : Int;   // Gapsize of this size parcel [cm]
   END_STRUCT;

END_TYPE

FUNCTION_BLOCK "FB_VfdNORDParaAcycRead"
{ S7_Optimized_Access := 'FALSE' }
VERSION : 0.1
// ATTRIBUTES
// AUTO_NUMBER = True
// BLOCK_NUMBER = 34
// END_ATTRIBUTES
   VAR_INPUT
      iHW_Identifier { ExternalAccessible := 'False'; ExternalVisible := 'False'; ExternalWritable := 'False'} : HW_IO;
      ii_FISystembus { ExternalAccessible := 'False'; ExternalVisible := 'False'; ExternalWritable := 'False'} : Int := 1;
      ii_Parameter_Number { ExternalAccessible := 'False'; ExternalVisible := 'False'; ExternalWritable := 'False'} : Int;
      ii_Parameter_Index { ExternalAccessible := 'False'; ExternalVisible := 'False'; ExternalWritable := 'False'} : Int;
      ii_Parameter_Set { ExternalAccessible := 'False'; ExternalVisible := 'False'; ExternalWritable := 'False'} : Int;
      ix_Enable { ExternalAccessible := 'False'; ExternalVisible := 'False'; ExternalWritable := 'False'} : Bool;
   END_VAR

   VAR_OUTPUT
      qdi_Value { ExternalAccessible := 'False'; ExternalVisible := 'False'; ExternalWritable := 'False'} : DInt;
      qw_Error_ID { ExternalAccessible := 'False'; ExternalVisible := 'False'; ExternalWritable := 'False'} : Word;
      qx_Valid { ExternalAccessible := 'False'; ExternalVisible := 'False'; ExternalWritable := 'False'} : Bool;
      qx_Busy { ExternalAccessible := 'False'; ExternalVisible := 'False'; ExternalWritable := 'False'} : Bool;
      qx_Error { ExternalAccessible := 'False'; ExternalVisible := 'False'; ExternalWritable := 'False'} : Bool;
   END_VAR

   VAR
      sa_Write_Val { ExternalAccessible := 'False'; ExternalVisible := 'False'; ExternalWritable := 'False'} : Array[0..3] of Word;
      sa_Rec_Write { ExternalAccessible := 'False'; ExternalVisible := 'False'; ExternalWritable := 'False'} AT sa_Write_Val : Struct
         PKE { ExternalAccessible := 'False'; ExternalVisible := 'False'; ExternalWritable := 'False'} : Word;
         Index { ExternalAccessible := 'False'; ExternalVisible := 'False'; ExternalWritable := 'False'} : Word;
         Para_Val { ExternalAccessible := 'False'; ExternalVisible := 'False'; ExternalWritable := 'False'} : DInt;
      END_STRUCT;
      sa_Read_Val { ExternalAccessible := 'False'; ExternalVisible := 'False'; ExternalWritable := 'False'} : Array[0..3] of Word;
      sa_Rec_Read { ExternalAccessible := 'False'; ExternalVisible := 'False'; ExternalWritable := 'False'} AT sa_Read_Val : Struct
         PKE { ExternalAccessible := 'False'; ExternalVisible := 'False'; ExternalWritable := 'False'} : Word;
         Index { ExternalAccessible := 'False'; ExternalVisible := 'False'; ExternalWritable := 'False'} : Word;
         Para_Val { ExternalAccessible := 'False'; ExternalVisible := 'False'; ExternalWritable := 'False'} : DInt;
      END_STRUCT;
      sv_WRREC_Instance {InstructionName := 'WRREC'; LibVersion := '1.1'; ExternalAccessible := 'False'; ExternalVisible := 'False'; ExternalWritable := 'False'; S7_SetPoint := 'False'} : WRREC;
      sv_RDREC_Instance {InstructionName := 'RDREC'; LibVersion := '1.0'; ExternalAccessible := 'False'; ExternalVisible := 'False'; ExternalWritable := 'False'; S7_SetPoint := 'False'} : RDREC;
      sw_Ak { ExternalAccessible := 'False'; ExternalVisible := 'False'; ExternalWritable := 'False'} : Word;
      sdi_Data_Record { ExternalAccessible := 'False'; ExternalVisible := 'False'; ExternalWritable := 'False'} : DInt;
      sdi_ValueStatic { ExternalAccessible := 'False'; ExternalVisible := 'False'; ExternalWritable := 'False'} : DInt;
      sw_Pnu { ExternalAccessible := 'False'; ExternalVisible := 'False'; ExternalWritable := 'False'} : Word;
      sw_ErrorIDStatic { ExternalAccessible := 'False'; ExternalVisible := 'False'; ExternalWritable := 'False'} : Word;
      si_Receivecounter { ExternalAccessible := 'False'; ExternalVisible := 'False'; ExternalWritable := 'False'} : Int;
      si_State { ExternalAccessible := 'False'; ExternalVisible := 'False'; ExternalWritable := 'False'} : Int;
      sx_ValidStatic { ExternalAccessible := 'False'; ExternalVisible := 'False'; ExternalWritable := 'False'} : Bool;
      sx_ErrorStatic { ExternalAccessible := 'False'; ExternalVisible := 'False'; ExternalWritable := 'False'} : Bool;
   END_VAR

   VAR_TEMP
      tw_ResponseIND : Word;
      tw_ResponseLABEL : Word;
      tw_ResponsePNU : Word;
      tdi_ResponsePWE : DInt;
      tx_WithIndex : Bool;
      tx_WithParameterSet : Bool;
   END_VAR

   VAR CONSTANT
      cw_IncorrectSubindex : Word := 3;
      cw_InternalResponseLabelCannotBeDepicted : Word := 202;
      cw_NoResponse : Word := 0;
      cw_OrderCannotBeExecuted : Word := 7;
      cw_OrderParameterValue : Word := 1;
      cw_ParameterOffset : Word := 1000;
      cw_PNUMask : Word := 16#07FF;
      ci_ReceivecounterMax : Int := 255;
      ci_Length : UInt := 8;
   END_VAR


BEGIN
	(*
	----------------------------------------------------------------------------------------

	Version history:
	Date        | Version   | Author        | Remark
	----------------------------------------------------------------------------------------
	25/01/2021  | 0.1       | S.Theocharis  | Copy from NORD library
	21/02/2023  | 4.0       | F.Baten       | 4.0 Release TIA 17.5
	*)

	#tx_WithIndex := #ii_Parameter_Index > 0;
	#tx_WithParameterSet := #ii_Parameter_Set > 0;

	CASE #si_State OF

	    0:
	        IF #ix_Enable AND
	            NOT ((#ii_Parameter_Set < 0) OR (#ii_Parameter_Index < 0) OR (#ii_Parameter_Set > 4) OR
	            (#tx_WithParameterSet AND (#ii_Parameter_Index > 64)) OR (NOT #tx_WithParameterSet AND (#ii_Parameter_Index > 256))) THEN
	            //initialize
	            #si_Receivecounter := 0;

	            // get PROFINET IO data record
	            IF (#ii_Parameter_Number >= 150 AND #ii_Parameter_Number <= 199) OR (#ii_Parameter_Number >= 800 AND #ii_Parameter_Number <= 849) THEN
	                // order to the bus interface
	                #sdi_Data_Record := 100;
	            ELSIF ((#ii_Parameter_Number >= 0 AND #ii_Parameter_Number < 150) OR (#ii_Parameter_Number >= 200 AND #ii_Parameter_Number <= 799) OR
	                (#ii_Parameter_Number >= 850 AND #ii_Parameter_Number <= 999)) AND (#ii_FISystembus > 0) AND (#ii_FISystembus <= 8) THEN
	                // order to frequency inverter 1..8
	                #sdi_Data_Record := #ii_FISystembus + 100;
	            ELSE
	                #sdi_Data_Record := 0;
	            END_IF;

	            // get order label (AK)
	            #sw_Ak := #cw_OrderParameterValue;

	            // merge parameter label (PKE)
	            #sw_Pnu := INT_TO_WORD(#ii_Parameter_Number + WORD_TO_INT(#cw_ParameterOffset));
	            #sa_Rec_Write.PKE := SHL(IN := #sw_Ak, N := 12) OR #sw_Pnu;

	            // get sub-index (IND)
	            IF #tx_WithIndex AND #tx_WithParameterSet THEN
	                #sa_Rec_Write.Index := SHL(IN := SHL(IN := INT_TO_WORD((#ii_Parameter_Index) - 1), N := 2) OR
	                                           INT_TO_WORD((#ii_Parameter_Set) - 1), N := 8);
	            ELSIF NOT #tx_WithIndex AND #tx_WithParameterSet THEN
	                #sa_Rec_Write.Index := SHL(IN := INT_TO_WORD((#ii_Parameter_Set) - 1), N := 8);
	            ELSIF #tx_WithIndex AND NOT #tx_WithParameterSet THEN
	                #sa_Rec_Write.Index := SHL(IN := INT_TO_WORD((#ii_Parameter_Index) - 1), N := 8);
	            ELSE
	                #sa_Rec_Write.Index := 0;
	            END_IF;

	            // check if parameter or index changed from last request
	            IF (#sa_Rec_Read.PKE AND #cw_PNUMask) <> (#sa_Rec_Write.PKE AND #cw_PNUMask) OR
	                (#sa_Rec_Read.Index <> #sa_Rec_Write.Index) THEN
	                // if changed reset valid bit
	                #sx_ValidStatic := FALSE;
	                #sx_ErrorStatic := FALSE;
	            END_IF;

	            // write data to device
	            #sv_WRREC_Instance(REQ := TRUE,
	                               ID := #iHW_Identifier,
	                               INDEX := #sdi_Data_Record,
	                               LEN := #ci_Length,
	                               DONE => #sv_WRREC_Instance.DONE,
	                               BUSY => #sv_WRREC_Instance.BUSY,
	                               ERROR => #sv_WRREC_Instance.ERROR,
	                               RECORD := #sa_Write_Val);
	            #si_State := 1;
	        ELSIF #ix_Enable AND
	            ((#ii_Parameter_Set < 0) OR (#ii_Parameter_Index < 0) OR (#ii_Parameter_Set > 4) OR
	            (#tx_WithParameterSet AND (#ii_Parameter_Index > 63)) OR (NOT #tx_WithParameterSet AND (#ii_Parameter_Index > 255))) THEN
	            #sx_ValidStatic := FALSE;
	            #sx_ErrorStatic := TRUE;
	            #sdi_ValueStatic := 0;
	            #sw_ErrorIDStatic := #cw_IncorrectSubindex;
	        ELSE
	            #sv_RDREC_Instance(REQ := FALSE,
	                               ID := #iHW_Identifier,
	                               INDEX := #sdi_Data_Record,
	                               MLEN := #ci_Length,
	                               RECORD := #sa_Read_Val);
	            #sx_ValidStatic := FALSE;
	            #sx_ErrorStatic := FALSE;
	            #sw_ErrorIDStatic := 0;
	            #sdi_ValueStatic := 0;
	        END_IF;

	    1:
	        #sv_WRREC_Instance();

	        IF #sv_WRREC_Instance.DONE THEN
	            #sv_WRREC_Instance(REQ := FALSE);
	            #si_State := 2;
	        ELSIF #sv_WRREC_Instance.ERROR THEN
	            #sx_ValidStatic := FALSE;
	            #sx_ErrorStatic := TRUE;
	            #sdi_ValueStatic := 0;
	            #sw_ErrorIDStatic := DWORD_TO_WORD(#sv_WRREC_Instance.STATUS);
	            #si_State := 0;
	        END_IF;

	    2:
	        #sv_RDREC_Instance(REQ := TRUE,
	                           ID := #iHW_Identifier,
	                           INDEX := #sdi_Data_Record,
	                           MLEN := #ci_Length,
	                           RECORD := #sa_Read_Val);

	        #tw_ResponseLABEL := SHR(IN := #sa_Rec_Read.PKE, N := 12);
	        #tw_ResponsePNU := #sa_Rec_Read.PKE AND #cw_PNUMask;
	        #tw_ResponseIND := #sa_Rec_Read.Index;
	        #tdi_ResponsePWE := #sa_Rec_Read.Para_Val;

	        IF #sv_RDREC_Instance.ERROR THEN
	            #sx_ValidStatic := FALSE;
	            #sx_ErrorStatic := TRUE;
	            #sdi_ValueStatic := 0;
	            #sw_ErrorIDStatic := DWORD_TO_WORD(#sv_RDREC_Instance.STATUS);
	            #si_State := 0;
	        ELSIF #sv_RDREC_Instance.VALID AND #tw_ResponseLABEL = #cw_OrderCannotBeExecuted THEN
	            #sx_ValidStatic := FALSE;
	            #sx_ErrorStatic := TRUE;
	            #sdi_ValueStatic := 0;
	            #sw_ErrorIDStatic := DINT_TO_WORD(#tdi_ResponsePWE);
	            #si_State := 0;
	        ELSIF #sv_RDREC_Instance.VALID AND #tw_ResponseLABEL <> #cw_NoResponse AND
	            #tw_ResponseLABEL <> #cw_OrderCannotBeExecuted AND #tw_ResponsePNU = #sw_Pnu AND
	            #tw_ResponseIND = #sa_Rec_Write.Index THEN
	            // acyclic read command complete
	            #sx_ValidStatic := TRUE;
	            #sx_ErrorStatic := FALSE;
	            #sdi_ValueStatic := #tdi_ResponsePWE;
	            #sw_ErrorIDStatic := 0;
	            #si_State := 0;
	        END_IF;

	        // check for read timeout
	        IF #si_Receivecounter >= #ci_ReceivecounterMax THEN
	            #sx_ValidStatic := FALSE;
	            #sx_ErrorStatic := TRUE;
	            #sdi_ValueStatic := 0;
	            #sw_ErrorIDStatic := #cw_InternalResponseLabelCannotBeDepicted;
	            #si_State := 0;
	        ELSE
	            #si_Receivecounter := #si_Receivecounter + 1;
	        END_IF;

	END_CASE;

	// output assignment
	#qx_Busy := INT_TO_BOOL(#si_State);
	IF #ix_Enable THEN
	    #qx_Valid := #sx_ValidStatic;
	    #qx_Error := #sx_ErrorStatic;
	    #qw_Error_ID := #sw_ErrorIDStatic;
	    #qdi_Value := #sdi_ValueStatic;
	ELSE
	    #qx_Valid := FALSE;
	    #qx_Error := FALSE;
	    #qw_Error_ID := 0;
	    #qdi_Value := 0;
	END_IF;
END_FUNCTION_BLOCK

FUNCTION_BLOCK "FB_VfdNORDParaAcycWrite"
{ S7_Optimized_Access := 'FALSE' }
VERSION : 0.1
// ATTRIBUTES
// AUTO_NUMBER = True
// BLOCK_NUMBER = 35
// END_ATTRIBUTES
   VAR_INPUT
      HW_Identifier { ExternalAccessible := 'False'; ExternalVisible := 'False'; ExternalWritable := 'False'} : HW_IO;
      idi_Value { ExternalAccessible := 'False'; ExternalVisible := 'False'; ExternalWritable := 'False'} : DInt;
      ii_FISystembus { ExternalAccessible := 'False'; ExternalVisible := 'False'; ExternalWritable := 'False'} : Int := 1;
      ii_ParameterNumber { ExternalAccessible := 'False'; ExternalVisible := 'False'; ExternalWritable := 'False'} : Int;
      ii_ParameterIndex { ExternalAccessible := 'False'; ExternalVisible := 'False'; ExternalWritable := 'False'} : Int;
      ii_ParameterSet { ExternalAccessible := 'False'; ExternalVisible := 'False'; ExternalWritable := 'False'} : Int;
      ix_Execute { ExternalAccessible := 'False'; ExternalVisible := 'False'; ExternalWritable := 'False'} : Bool;
      ix_Parameter32Bit { ExternalAccessible := 'False'; ExternalVisible := 'False'; ExternalWritable := 'False'} : Bool;
      ix_RAM_Only { ExternalAccessible := 'False'; ExternalVisible := 'False'; ExternalWritable := 'False'} : Bool;
   END_VAR

   VAR_OUTPUT
      qx_Done { ExternalAccessible := 'False'; ExternalVisible := 'False'; ExternalWritable := 'False'} : Bool;
      qx_Busy { ExternalAccessible := 'False'; ExternalVisible := 'False'; ExternalWritable := 'False'} : Bool;
      qx_Error { ExternalAccessible := 'False'; ExternalVisible := 'False'; ExternalWritable := 'False'} : Bool;
      qdi_ValueRead { ExternalAccessible := 'False'; ExternalVisible := 'False'; ExternalWritable := 'False'} : DInt;
      qw_ErrorID { ExternalAccessible := 'False'; ExternalVisible := 'False'; ExternalWritable := 'False'} : Word;
   END_VAR

   VAR
      sa_WriteVal { ExternalAccessible := 'False'; ExternalVisible := 'False'; ExternalWritable := 'False'} : Array[0..3] of Word;
      sa_RecWrite { ExternalAccessible := 'False'; ExternalVisible := 'False'; ExternalWritable := 'False'} AT sa_WriteVal : Struct
         PKE { ExternalAccessible := 'False'; ExternalVisible := 'False'; ExternalWritable := 'False'} : Word;
         Index { ExternalAccessible := 'False'; ExternalVisible := 'False'; ExternalWritable := 'False'} : Word;
         Para_Val { ExternalAccessible := 'False'; ExternalVisible := 'False'; ExternalWritable := 'False'} : DInt;
      END_STRUCT;
      sa_ReadVal { ExternalAccessible := 'False'; ExternalVisible := 'False'; ExternalWritable := 'False'} : Array[0..3] of Word;
      sa_RecRead { ExternalAccessible := 'False'; ExternalVisible := 'False'; ExternalWritable := 'False'} AT sa_ReadVal : Struct
         PKE { ExternalAccessible := 'False'; ExternalVisible := 'False'; ExternalWritable := 'False'} : Word;
         Index { ExternalAccessible := 'False'; ExternalVisible := 'False'; ExternalWritable := 'False'} : Word;
         Para_Val { ExternalAccessible := 'False'; ExternalVisible := 'False'; ExternalWritable := 'False'} : DInt;
      END_STRUCT;
      sv_WRRECInstance {InstructionName := 'WRREC'; LibVersion := '1.1'; ExternalAccessible := 'False'; ExternalVisible := 'False'; ExternalWritable := 'False'; S7_SetPoint := 'False'} : WRREC;
      sv_RDRECInstance {InstructionName := 'RDREC'; LibVersion := '1.0'; ExternalAccessible := 'False'; ExternalVisible := 'False'; ExternalWritable := 'False'; S7_SetPoint := 'False'} : RDREC;
      sw_Ak { ExternalAccessible := 'False'; ExternalVisible := 'False'; ExternalWritable := 'False'} : Word;
      sw_Pnu { ExternalAccessible := 'False'; ExternalVisible := 'False'; ExternalWritable := 'False'} : Word;
      sw_ErrorIDStatic { ExternalAccessible := 'False'; ExternalVisible := 'False'; ExternalWritable := 'False'} : Word;
      sdi_DataRecord { ExternalAccessible := 'False'; ExternalVisible := 'False'; ExternalWritable := 'False'} : DInt;
      si_Receivecounter { ExternalAccessible := 'False'; ExternalVisible := 'False'; ExternalWritable := 'False'} : Int;
      si_State { ExternalAccessible := 'False'; ExternalVisible := 'False'; ExternalWritable := 'False'} : Int;
      sx_FLMExecute { ExternalAccessible := 'False'; ExternalVisible := 'False'; ExternalWritable := 'False'} : Bool;
      sx_REdgeExecute { ExternalAccessible := 'False'; ExternalVisible := 'False'; ExternalWritable := 'False'} : Bool;
      sx_DoneStatic { ExternalAccessible := 'False'; ExternalVisible := 'False'; ExternalWritable := 'False'} : Bool;
      sx_ErrorStatic { ExternalAccessible := 'False'; ExternalVisible := 'False'; ExternalWritable := 'False'} : Bool;
   END_VAR

   VAR_TEMP
      tw_ResponseIND : Word;
      tw_ResponseLABEL : Word;
      tw_ResponsePNU : Word;
      tdi_ResponsePWE : DInt;
      tx_WithIndex : Bool;
      tx_WithParameterSet : Bool;
   END_VAR

   VAR CONSTANT
      cw_ChangeParameterValueWordEEPROM : Word := 2;
      cw_ChangeParameterValueWordRAM : Word := 14;
      cw_ChangeParameterValueDoubleWordEEPROM : Word := 3;
      cw_ChangeParameterValueDoubleWordRAM : Word := 13;
      cw_IncorretSubindex : Word := 3;
      cw_InternalResponseLabelCannotBeDepicted : Word := 202;
      cw_InvalidDataType : Word := 5;
      cw_NoResponse : Word := 0;
      cw_OrderCannotBeExecuted : Word := 7;
      cw_ParameterOffset : Word := 1000;
      cw_PNUMask : Word := 16#07FF;
      ci_ReceivecounterMax : Int := 255;
      ci_Length : UInt := 8;
   END_VAR


BEGIN
	(*
	----------------------------------------------------------------------------------------

	Version history:
	Date        | Version   | Author        | Remark
	----------------------------------------------------------------------------------------
	25/01/2021  | 0.1       | S.Theocharis  | Copy fron NORD library
	21/02/2023  | 4.0       | F.Baten       | 4.0 Release TIA 17.5
	*)
	// protects the frequency inverter from too frequent write requests.
	IF #ix_Execute <> #sx_FLMExecute THEN
	    IF #ix_Execute THEN
	        #sx_REdgeExecute := TRUE;
	    ELSE
	        #sx_REdgeExecute := FALSE;
	    END_IF;
	    #sx_FLMExecute := #ix_Execute;
	ELSE
	    #sx_REdgeExecute := FALSE;
	END_IF;

	#tx_WithIndex := #ii_ParameterIndex > 0;
	#tx_WithParameterSet := #ii_ParameterSet > 0;

	CASE #si_State OF

	    0:
	        IF #sx_REdgeExecute AND
	            NOT ((#ii_ParameterSet < 0) OR (#ii_ParameterIndex < 0) OR (#ii_ParameterSet > 4) OR
	            (#tx_WithParameterSet AND (#ii_ParameterIndex > 64)) OR (NOT #tx_WithParameterSet AND (#ii_ParameterIndex > 256)) OR
	            (NOT #ix_Parameter32Bit AND #idi_Value < -32768) OR (NOT #ix_Parameter32Bit AND #idi_Value > 16#FFFF)) THEN
	            //initialize
	            #sx_DoneStatic := FALSE;
	            #sx_ErrorStatic := FALSE;
	            #sw_ErrorIDStatic := 0;
	            #si_Receivecounter := 0;
	            #qx_Done := FALSE;
	            #qx_Busy := TRUE;

	            // get PROFINET IO data record
	            IF (#ii_ParameterNumber >= 150 AND #ii_ParameterNumber <= 199) OR (#ii_ParameterNumber >= 800 AND #ii_ParameterNumber <= 849) THEN
	                // order to the bus interface
	                #sdi_DataRecord := 100;
	            ELSIF ((#ii_ParameterNumber >= 0 AND #ii_ParameterNumber < 150) OR (#ii_ParameterNumber >= 200 AND #ii_ParameterNumber <= 799) OR
	                (#ii_ParameterNumber >= 850 AND #ii_ParameterNumber <= 999)) AND (#ii_FISystembus > 0) AND (#ii_FISystembus <= 8) THEN
	                // order to frequency inverter 1..8
	                #sdi_DataRecord := #ii_FISystembus + 100;
	            ELSE
	                #sdi_DataRecord := 0;
	            END_IF;

	            // get order label (AK)
	            IF #ix_RAM_Only THEN
	                IF #ix_Parameter32Bit THEN
	                    #sw_Ak := #cw_ChangeParameterValueDoubleWordRAM;
	                ELSE
	                    #sw_Ak := #cw_ChangeParameterValueWordRAM;
	                END_IF;
	            ELSE
	                IF #ix_Parameter32Bit THEN
	                    #sw_Ak := #cw_ChangeParameterValueDoubleWordEEPROM;
	                ELSE
	                    #sw_Ak := #cw_ChangeParameterValueWordEEPROM;
	                END_IF;
	            END_IF;

	            // merge parameter label (PKE)
	            #sw_Pnu := INT_TO_WORD(#ii_ParameterNumber + WORD_TO_INT(#cw_ParameterOffset));
	            #sa_RecWrite.PKE := SHL(IN := #sw_Ak, N := 12) OR #sw_Pnu;

	            // get sub-index (IND)
	            IF #tx_WithIndex AND #tx_WithParameterSet THEN
	                #sa_RecWrite.Index := SHL(IN := SHL(IN := INT_TO_WORD((#ii_ParameterIndex) - 1), N := 2) OR
	                                          INT_TO_WORD((#ii_ParameterSet) - 1), N := 8);
	            ELSIF NOT #tx_WithIndex AND #tx_WithParameterSet THEN
	                #sa_RecWrite.Index := SHL(IN := INT_TO_WORD((#ii_ParameterSet) - 1), N := 8);
	            ELSIF #tx_WithIndex AND NOT #tx_WithParameterSet THEN
	                #sa_RecWrite.Index := SHL(IN := INT_TO_WORD((#ii_ParameterIndex) - 1), N := 8);
	            ELSE
	                #sa_RecWrite.Index := 0;
	            END_IF;

	            // get parameter value (PWE)
	            #sa_RecWrite.Para_Val := #idi_Value;

	            // write data to device
	            #sv_WRRECInstance(REQ := TRUE,
	                              ID := #HW_Identifier,
	                              INDEX := #sdi_DataRecord,
	                              LEN := #ci_Length,
	                              DONE => #sv_WRRECInstance.DONE,
	                              BUSY => #sv_WRRECInstance.BUSY,
	                              ERROR => #sv_WRRECInstance.ERROR,
	                              RECORD := #sa_WriteVal);
	            #si_State := 1;
	        ELSIF #sx_REdgeExecute AND
	            ((#ii_ParameterSet < 0) OR (#ii_ParameterIndex < 0) OR (#ii_ParameterSet > 4) OR
	            (#tx_WithParameterSet AND (#ii_ParameterIndex > 63)) OR (NOT #tx_WithParameterSet AND (#ii_ParameterIndex > 255))) THEN
	            #sx_DoneStatic := FALSE;
	            #sx_ErrorStatic := TRUE;
	            #sw_ErrorIDStatic := #cw_IncorretSubindex;
	        ELSIF #sx_REdgeExecute AND
	            ((NOT #ix_Parameter32Bit AND #idi_Value < -32768) OR (NOT #ix_Parameter32Bit AND #idi_Value > 16#FFFF)) THEN
	            // limitation to int value range. positive hex crc checksums are allowed
	            #sx_DoneStatic := FALSE;
	            #sx_ErrorStatic := TRUE;
	            #sw_ErrorIDStatic := #cw_InvalidDataType;
	        ELSE
	            #sv_RDRECInstance(REQ := FALSE,
	                              ID := #HW_Identifier,
	                              INDEX := #sdi_DataRecord,
	                              MLEN := #ci_Length,
	                              RECORD := #sa_ReadVal);
	        END_IF;

	    1:
	        #sv_WRRECInstance();

	        IF #sv_WRRECInstance.DONE THEN
	            #sv_WRRECInstance(REQ := FALSE);
	            #si_State := 2;
	        ELSIF #sv_WRRECInstance.ERROR THEN
	            #sx_DoneStatic := FALSE;
	            #sx_ErrorStatic := TRUE;
	            #sw_ErrorIDStatic := DWORD_TO_WORD(#sv_WRRECInstance.STATUS);
	            #si_State := 0;
	            #qx_Done := FALSE;
	            #qx_Busy := TRUE;
	        END_IF;

	    2:
	        #sv_RDRECInstance(REQ := TRUE,
	                          ID := #HW_Identifier,
	                          INDEX := #sdi_DataRecord,
	                          MLEN := #ci_Length,
	                          RECORD := #sa_ReadVal);

	        #tw_ResponseLABEL := SHR(IN := #sa_RecRead.PKE, N := 12);
	        #tw_ResponsePNU := #sa_RecRead.PKE AND #cw_PNUMask;
	        #tw_ResponseIND := #sa_RecRead.Index;
	        #tdi_ResponsePWE := #sa_RecRead.Para_Val;
	        #qdi_ValueRead := #sa_RecRead.Para_Val;
	        IF #sv_RDRECInstance.ERROR THEN
	            #sx_DoneStatic := FALSE;
	            #sx_ErrorStatic := TRUE;
	            #sw_ErrorIDStatic := DWORD_TO_WORD(#sv_RDRECInstance.STATUS);
	            #si_State := 0;
	        ELSIF #sv_RDRECInstance.VALID AND #tw_ResponseLABEL = #cw_OrderCannotBeExecuted THEN
	            #sx_DoneStatic := FALSE;
	            #sx_ErrorStatic := TRUE;
	            #sw_ErrorIDStatic := DINT_TO_WORD(#tdi_ResponsePWE);
	            #si_State := 0;
	        ELSIF #sv_RDRECInstance.VALID AND #tw_ResponseLABEL <> #cw_NoResponse AND
	            #tw_ResponseLABEL <> #cw_OrderCannotBeExecuted AND #tw_ResponsePNU = #sw_Pnu AND
	            #tw_ResponseIND = #sa_RecWrite.Index THEN
	            // acyclic write command complete
	            #sx_DoneStatic := TRUE;
	            #si_State := 0;
	        END_IF;

	        // check for read timeout
	        IF #si_Receivecounter >= #ci_ReceivecounterMax THEN
	            #sx_DoneStatic := FALSE;
	            #sx_ErrorStatic := TRUE;
	            #sw_ErrorIDStatic := #cw_InternalResponseLabelCannotBeDepicted;
	            #si_State := 0;
	        ELSE
	            #si_Receivecounter := #si_Receivecounter + 1;
	        END_IF;
	END_CASE;

	// output assignment
	#qx_Busy := INT_TO_BOOL(#si_State) AND NOT #sx_DoneStatic AND NOT #sx_ErrorStatic;
	IF #ix_Execute THEN
	    #qx_Done := #sx_DoneStatic;
	    #qx_Error := #sx_ErrorStatic;
	    #qw_ErrorID := #sw_ErrorIDStatic;
	ELSE
	    #qx_Done := FALSE;
	    #qx_Error := FALSE;
	    #qw_ErrorID := 0;
	END_IF;
END_FUNCTION_BLOCK

TYPE "UDT_VfdNordParameter"
TITLE = UDT_VfdNordParameter
VERSION : 0.1
//Parameter structure to read and write
   STRUCT
      WriteValue : DInt;   // Parameter value to write
      ActualValue : DInt;   // Actual value read from VFD
      ParaNumber : Int;   // Parameter number to access
      Index : Int;   // Parameter index number to access
      ParaSet : Int;   // Parameter set to acces
      Format32 { ExternalAccessible := 'False'; ExternalVisible := 'False'; ExternalWritable := 'False'} : Bool;   // 1 = Write the parameter in DWord format. 0 = Write the parameter in Word format
      WriteAccess { ExternalAccessible := 'False'; ExternalVisible := 'False'; ExternalWritable := 'False'} : Bool;   // 1 = Write the parameter. 0 = Read the parameter
      InUse { ExternalAccessible := 'False'; ExternalVisible := 'False'; ExternalWritable := 'False'} : Bool;   // 1 = Parameter is to be processed
      RamOnly { ExternalAccessible := 'False'; ExternalVisible := 'False'; ExternalWritable := 'False'} : Bool;   // 1 = Save parameter in RAM, 0 = Save parameter in RAM and EEPROM
   END_STRUCT;

END_TYPE

TYPE "UDT_FifoHeader"
TITLE = UDT_FifoHeader
VERSION : 0.1
//User-defined structure of FIFO register header information.
   STRUCT
      Status : Struct   // Status bits
         Empty { ExternalAccessible := 'False'; ExternalVisible := 'False'; ExternalWritable := 'False'} : Bool;   // FIFO Empty
         Prefull { ExternalAccessible := 'False'; ExternalVisible := 'False'; ExternalWritable := 'False'} : Bool;   // FIFO Prefull
         Full { ExternalAccessible := 'False'; ExternalVisible := 'False'; ExternalWritable := 'False'} : Bool;   // FIFO Full
      END_STRUCT;
      NextEntryToRead : Int;   // Next FIFO entry to read
      NextEntryToWrite : Int;   // Next FIFO entry to write
      MaxNrOfEntries : Int;   // Maximum number of FIFO entries
      TotalEntriesStored : Int;   // Total number of FIFO entries
   END_STRUCT;

END_TYPE

TYPE "UDT_FIFOInductInfo"
VERSION : 0.1
   STRUCT
      InductNumber : Int;   // Induct number
      GapSize : Int;   // Size of gap requested by induct
      RemoveEntry { ExternalAccessible := 'False'; ExternalVisible := 'False'; ExternalWritable := 'False'} : Bool;   // Entry is not needed by induct anymore
   END_STRUCT;

END_TYPE

TYPE "UDT_FifoStatus"
TITLE = UDT_FifoStatus
VERSION : 0.1
//
//User-defined structure of FC_Fifo function status.
//Version History:
//Date              | Version   | Author         | Remark
//24/05/2019  | 0.1           | K.Pokorski   | first release MHSE TIA 15.1
//24/05/2019  | 0.2           | K.Pokorski   | first release MHSE TIA 15.1
//
   STRUCT
      InvalidMode { ExternalAccessible := 'False'; ExternalVisible := 'False'; ExternalWritable := 'False'} : Bool;   // Invalid mode selected
      InvalidMaxNrOfEntries { ExternalAccessible := 'False'; ExternalVisible := 'False'; ExternalWritable := 'False'} : Bool;   // Invalid maximum number of entries or buffer is not an array
      InvalidTotalEntriesStored { ExternalAccessible := 'False'; ExternalVisible := 'False'; ExternalWritable := 'False'} : Bool;   // Invalid total number of entries
      InvalidNextEntryToWrite { ExternalAccessible := 'False'; ExternalVisible := 'False'; ExternalWritable := 'False'} : Bool;   // Invalid number of next entry to write
      InvalidNextEntryToRead { ExternalAccessible := 'False'; ExternalVisible := 'False'; ExternalWritable := 'False'} : Bool;   // Invalid number of next entry to read
      InvalidDataType { ExternalAccessible := 'False'; ExternalVisible := 'False'; ExternalWritable := 'False'} : Bool;   // Message and buffer element data type inconsistent
      FifoPreFull { ExternalAccessible := 'False'; ExternalVisible := 'False'; ExternalWritable := 'False'} : Bool;   // 90 % of FIFO data buffer capacity reached
      FifoFull { ExternalAccessible := 'False'; ExternalVisible := 'False'; ExternalWritable := 'False'} : Bool;   // FIFO data buffer full
   END_STRUCT;

END_TYPE

DATA_BLOCK "DB_GIN"
TITLE = DB_GIN
{ S7_Optimized_Access := 'TRUE' }
AUTHOR : MHSE
FAMILY : GeneralSystemFunctions
VERSION : 3.0
NON_RETAIN
//Data block to store parcels informations.
   VAR
      GIN { ExternalAccessible := 'False'; ExternalVisible := 'False'; ExternalWritable := 'False'; S7_SetPoint := 'False'} : Array[1..1] of "UDT_GIN";   // GIN informations - for project remove unneeded customers and extend array bound range to 9999
   END_VAR


BEGIN

END_DATA_BLOCK

DATA_BLOCK "DB_HMIStatusConfiguration"
TITLE = DB_HMIStatusConfiguration
{ S7_Optimized_Access := 'TRUE' }
AUTHOR : MHSE
VERSION : 3.0
NON_RETAIN
   VAR
      FireAlarm : Int;   // Fire alarm active
      SafetyStop : Int;   // Safety stop error status
      Error : Int;   // Error status
      Warning : Int;   // Warning status
      ManualRun : Int;   // Manual run status
      Manual : Int;   // Manual status
      Halted : Int;   // Halted status
      Dieback : Int;   // Die back status
      Stopped : Int;   // Stopped status
      Running : Int;   // Running status
      EnergySave : Int;   // Energy save status
      CommunicationError : Int;   // Communication error status
      CBError : Int;   // CB error status
      ProfinetError : Int;   // Profinet error status
      HardwareError : Int;   // Hardware error status
      VFDNotHealthy : Int;   // VFD noth healthy status
      VFDError : Int;   // VFD error status
      PECJam : Int;   // PEC jam status
      ChuteFull : Int;   // Chute full status
      EncoderError : Int;   // Encoder error status
      TrackingError : Int;   // Tracking error status
      DimensionError : Int;   // Dimension error status
      OperationalError : Int;   // Operational error status
      AutoON : Int;   // Automatic is on
      ChuteHalfFull : Int;   // Disable by operator
      DisableByManagement : Int;   // Disable by management
      GateOpen : Int;   // Manual operated gate is open
      GateClosed : Int;   // Manual operated gate is closed
      GateClosedAndNoOperatorPresent : Int;   // Manual operated gate is closed and no operator is present
      PositionChangeOngoing : Int;   // Lifting device or arm diverter changing position
      BufferMode : Int;   // BufferMode Active
      ContinuousMode : Int;   // ContinuousMode Active
      LabbelingMode : Int;   // LabbelingMode Active
   END_VAR


BEGIN
   FireAlarm := 1;
   SafetyStop := 3;
   Error := 5;
   Warning := 7;
   ManualRun := 9;
   Manual := 11;
   Halted := 13;
   Dieback := 15;
   Stopped := 17;
   Running := 19;
   EnergySave := 21;
   CommunicationError := 23;
   CBError := 25;
   ProfinetError := 27;
   HardwareError := 29;
   VFDNotHealthy := 31;
   VFDError := 33;
   PECJam := 35;
   ChuteFull := 37;
   EncoderError := 39;
   TrackingError := 41;
   DimensionError := 43;
   OperationalError := 45;
   AutoON := 47;
   ChuteHalfFull := 49;
   DisableByManagement := 51;
   GateOpen := 53;
   GateClosed := 55;
   GateClosedAndNoOperatorPresent := 57;
   PositionChangeOngoing := 59;
   BufferMode := 61;
   ContinuousMode := 63;
   LabbelingMode := 65;

END_DATA_BLOCK

FUNCTION_BLOCK "FB_TimerOnOffDelay"
TITLE = FB_TimerOnOffDelay
{ S7_Optimized_Access := 'TRUE' }
AUTHOR : MHSE
FAMILY : GeneralSystemFunctions
VERSION : 3.0
// ATTRIBUTES
// AUTO_NUMBER = True
// BLOCK_NUMBER = 32
// END_ATTRIBUTES
//Function block to generate on/off signal delay.
   VAR_INPUT
      iudi_OnDelayTime { ExternalAccessible := 'False'; ExternalVisible := 'False'; ExternalWritable := 'False'} : UDInt;   // On delay time [ms]
      iudi_OffDelayTime { ExternalAccessible := 'False'; ExternalVisible := 'False'; ExternalWritable := 'False'} : UDInt;   // Off delay time [ms]
      ix_SignalToDelay { ExternalAccessible := 'False'; ExternalVisible := 'False'; ExternalWritable := 'False'} : Bool;   // Input signal to be delayed
      ix_Enable { ExternalAccessible := 'False'; ExternalVisible := 'False'; ExternalWritable := 'False'} : Bool := TRUE;   // Timer Enable
   END_VAR

   VAR_OUTPUT
      qlr_ActualTime { ExternalAccessible := 'False'; ExternalVisible := 'False'; ExternalWritable := 'False'} : LReal;   // Actual time
      qx_DelayedSignal { ExternalAccessible := 'False'; ExternalVisible := 'False'; ExternalWritable := 'False'} : Bool;   // Delayed signal output
   END_VAR

   VAR
      s_R_TRIG_Signal {InstructionName := 'R_TRIG'; LibVersion := '1.0'; ExternalAccessible := 'False'; ExternalVisible := 'False'; ExternalWritable := 'False'; S7_SetPoint := 'False'} : R_TRIG;   // Siemens "R_Trig" - to prepare the rising edge trigger on "ix_SignalToDelay" signal
      s_F_TRIG_Signal {InstructionName := 'F_TRIG'; LibVersion := '1.0'; ExternalAccessible := 'False'; ExternalVisible := 'False'; ExternalWritable := 'False'; S7_SetPoint := 'False'} : F_TRIG;   // Siemens "F_Trig" - to prepare the falling edge trigger on "ix_SignalToDelay" signal
   END_VAR
   VAR RETAIN
      slr_ActualDelayTime { ExternalAccessible := 'False'; ExternalVisible := 'False'; ExternalWritable := 'False'} : LReal;   // Actual delay time [ms]
   END_VAR


BEGIN
	(*
	----------------------------------------------------------------------------------------

	Version history:
	Date        | Version   | Author        | Remark
	----------------------------------------------------------------------------------------
	24/05/2019  | 0.1       | L.Klar        | first release MHS TIA 15.1
	24/07/2019  | 2.0       | L.Klar        | 2.0 MHS library release TIA 15.1
	26/08/2019  | 2.1       | M.Kurpiers    | Comments adjusted
	04/11/2019  | 2.2       | L.Klar        | Prevoius cycle scan changed from memory to DB variable
	12/11/2019  | 3.0       | P.Majka       | 3.0 MHS library release TIA 15.1
	21/02/2023  | 4.0       | F.Baten       | 4.0 Release TIA 17.5
	*)

	REGION Step 1 – Input signal edge detection

	    #s_R_TRIG_Signal(CLK := #ix_SignalToDelay);


	    #s_F_TRIG_Signal(CLK := #ix_SignalToDelay);

	END_REGION

	REGION Step 2 – Actual delay time initialization

	    IF (#s_R_TRIG_Signal.Q OR #s_F_TRIG_Signal.Q)           // Input signal changed
	    THEN

	        #slr_ActualDelayTime := 0;

	    END_IF;

	END_REGION

	REGION Step 3 – On/Off delay time calculation


	    IF (#ix_SignalToDelay                                       // Signal to be delayed is active
	        AND #ix_Enable)                                         // Ttimer enabled
	    THEN

	        // Timer on
	        IF (#slr_ActualDelayTime >= #iudi_OnDelayTime)
	        THEN

	            #qx_DelayedSignal := TRUE;

	        ELSE

	            #slr_ActualDelayTime += "DB_Memory".PrevCycleTime;

	        END_IF;

	    END_IF;

	    // Timer off
	    IF (NOT #ix_SignalToDelay                                   // Signal to delay is not active
	        AND #ix_Enable)                                         // Timer is enabled
	    THEN

	        IF (#slr_ActualDelayTime >= #iudi_OffDelayTime)
	        THEN

	            #qx_DelayedSignal := FALSE;

	        ELSE

	            #slr_ActualDelayTime += "DB_Memory".PrevCycleTime;

	        END_IF;

	    END_IF;

	END_REGION

	REGION Step 4 – Actual time

	    #qlr_ActualTime := #slr_ActualDelayTime;

	END_REGION
END_FUNCTION_BLOCK

TYPE "UDT_PECConfiguration"
VERSION : 0.1
   STRUCT
      Distance : DInt;   // Distance between photo eye and the end of conveyor [mm]
      JamDisplacementLimit : Int;   // Limit displacement with PEC blocked o detect jam [cm]
      TimeOnDelay : UDInt;   // Photo eye time on delay [ms]
      TimeOffDelay : UDInt;   // Photo eye time off delay [ms]
      ResetWithPECBlocked { ExternalAccessible := 'False'; ExternalVisible := 'False'; ExternalWritable := 'False'} : Bool;   // When 'True' Allow reset system after jam with PEC blocked
   END_STRUCT;

END_TYPE

TYPE "UDT_ConveyorHandshake"
TITLE = UDT_ConveyorHandshake
VERSION : 0.1
//User-defined structure of conveyor handshake variables.
   STRUCT
      GIN : Int;   // General identification number
      NrOfPosToShift : Int;   // Number of positions to shift
      DownstreamDisplacement : Int;   // Displacement from downstream [cm]
      RTS { ExternalAccessible := 'False'; ExternalVisible := 'False'; ExternalWritable := 'False'} : Bool;   // Conveyor ready to send
      RTR { ExternalAccessible := 'False'; ExternalVisible := 'False'; ExternalWritable := 'False'} : Bool;   // Conveyor ready to receive
      TIP { ExternalAccessible := 'False'; ExternalVisible := 'False'; ExternalWritable := 'False'} : Bool;   // Transfer in progress
      ResetEnergySave { ExternalAccessible := 'False'; ExternalVisible := 'False'; ExternalWritable := 'False'} : Bool;   // Reset energy save mode
      CascadeStartUp { ExternalAccessible := 'False'; ExternalVisible := 'False'; ExternalWritable := 'False'} : Bool;   // Cascade startup
      ReqStop { ExternalAccessible := 'False'; ExternalVisible := 'False'; ExternalWritable := 'False'} : Bool;   // Request stop
   END_STRUCT;

END_TYPE

TYPE "UDT_AixControllerStatus"
VERSION : 0.1
   STRUCT
      MotorStatus { ExternalWritable := 'False'; S7_SetPoint := 'False'} : "UDT_AixMotorStatus";
      SpeedFeedbackError { ExternalAccessible := 'False'; ExternalVisible := 'False'; ExternalWritable := 'False'} : Bool;   // TRUE if  right motor deviates from set speed
      InternalWarning { ExternalWritable := 'False'} : Bool := FALSE;   // An internal warning is active
      InternalError { ExternalAccessible := 'False'; ExternalVisible := 'False'; ExternalWritable := 'False'} : Bool;   // An internal error is active
      CommunicationErrorVFD { ExternalAccessible := 'False'; ExternalVisible := 'False'; ExternalWritable := 'False'} : Bool;   // Communication with VFD timed out
      PNSlaveNotOnline { ExternalWritable := 'False'} : Bool := FALSE;   // Profinet slave is not on line
      PNSlaveError { ExternalWritable := 'False'} : Bool := FALSE;   // Profinet slave has an error
      PNSlaveWarning { ExternalWritable := 'False'} : Bool := FALSE;   // Profinet slave has a warning
      ControllerStatus : DWord;
   END_STRUCT;

END_TYPE

TYPE "UDT_GOSLog"
VERSION : 0.1
   STRUCT
      GIN_nr : Int;
      InfeedUpstreamGap : Int;   // Gap in millimeters (mm)
      InfeedDownstreamGap : Int;   // Gap in millimeters (mm)
      OutfeedUpstreamGap : Int;   // Gap in meters (mm)
      OutfeedDownstreamGap : Int;   // Gap in meters (mm)
      ParcelLength : Int;
      GapToBeRecovered : Int;
      ParcelDownStreamResults : Int;
      ParcelUpStreamResults : Int;
      Accelerate { ExternalAccessible := 'False'; ExternalVisible := 'False'; ExternalWritable := 'False'} : Bool;
      Decelerate { ExternalAccessible := 'False'; ExternalVisible := 'False'; ExternalWritable := 'False'} : Bool;
      PrevConveyorUpstreamGap : Int;
      PrevConveyorDownstreamGap : Int;
      NextConveyorUpstreamGap : Int;
      NextConveyorDownstreamGap : Int;
   END_STRUCT;

END_TYPE

TYPE "UDT_PECStatus"
VERSION : 0.1
   STRUCT
      PEC { ExternalAccessible := 'False'; ExternalVisible := 'False'; ExternalWritable := 'False'} : Bool;   // Current state of the photo eye
      Jam { ExternalAccessible := 'False'; ExternalVisible := 'False'; ExternalWritable := 'False'} : Bool;   // PEC jam error
   END_STRUCT;

END_TYPE

FUNCTION "FC_Statistics" : Void
TITLE = FC_Statistics
{ S7_Optimized_Access := 'TRUE' }
AUTHOR : MHSE
FAMILY : GeneralSystemFunctions
VERSION : 3.0
// ATTRIBUTES
// AUTO_NUMBER = True
// BLOCK_NUMBER = 26
// END_ATTRIBUTES
//Function to calculate statistics.
   VAR_INPUT
      ix_Reset : Bool;   // Reset statistics data
      ix_Activate : Bool;   // Activete statistics counters
      ix_RTrigActivate : Bool;   // Activation rise trigger
   END_VAR

   VAR_IN_OUT
      iqUDT_Statistics : "UDT_EventStatistic";   // Statistic structure
   END_VAR


BEGIN
	(*
	----------------------------------------------------------------------------------------

	Version history:
	Date        | Version   | Author        | Remark
	----------------------------------------------------------------------------------------
	24/05/2019  | 0.1       | C. Leite      | first release MHS TIA 15.1
	17/07/2019  | 0.2       | A.Nowak       | Add comments
	24/07/2019  | 2.0       | L.Klar        | 2.0 MHS library release TIA 15.1
	27/08/2019  | 2.1       | M.Kurpiers    | Comments adjusted
	04/11/2019  | 2.2       | L.Klar        | 1 second pulse changed from memory bit to DB variable
	12/11/2019  | 3.0       | P.Majka       | 3.0 MHS library release TIA 15.1
	21/02/2023  | 4.0       | F.Baten       | 4.0 Release TIA 17.5
	*)

	REGION 1 - Number of events

	    IF (#ix_RTrigActivate)      // Event occured
	    THEN

	        // Increment the number of times the event occurred and clear the time of the current or last event
	        #iqUDT_Statistics.NumberOfTimes += 1;
	        #iqUDT_Statistics.LastEventSeconds := 0;

	    END_IF;

	END_REGION

	REGION 2 - Event time

	    // 1 shot every 1 sec and activate statistic counter
	    IF ("DB_Memory".OS_1sec AND #ix_Activate)
	    THEN

	        // Increment the time of the current or last event and the time of all events that occured
	        #iqUDT_Statistics.LastEventSeconds += 1;
	        #iqUDT_Statistics.TotalEventSeconds += 1;

	    END_IF;

	END_REGION

	REGION 3 - Data reset


	    IF (#ix_Reset)                                            // Reset statistics data
	    THEN

	        IF (NOT #ix_Activate)                                 // Statistic counter isn't activate
	        THEN

	            // Clear statistics data
	            #iqUDT_Statistics.NumberOfTimes := 0;
	            #iqUDT_Statistics.LastEventSeconds := 0;
	            #iqUDT_Statistics.TotalEventSeconds := 0;

	        ELSE

	            // Write 1 to the number of times the event occurred and clear times
	            #iqUDT_Statistics.NumberOfTimes := 1;
	            #iqUDT_Statistics.LastEventSeconds := 0;
	            #iqUDT_Statistics.TotalEventSeconds := 0;

	        END_IF;

	    END_IF;

	END_REGION
END_FUNCTION

TYPE "UDT_PECStatistics"
VERSION : 0.1
   STRUCT
      Jam : "UDT_EventStatistic";   // Number of times PEC got jammed
   END_STRUCT;

END_TYPE

TYPE "UDT_RIOStatus"
VERSION : 0.1
   STRUCT
      Status : Int;   // Status number
      Specific : Struct   // Specific structure
         PNSlaveNotOnline { ExternalAccessible := 'False'; ExternalVisible := 'False'; ExternalWritable := 'False'} : Bool;   // Profinet slave is not online
         PNSlaveError { ExternalAccessible := 'False'; ExternalVisible := 'False'; ExternalWritable := 'False'} : Bool;   // Profinet slave is in error
         ET200sp_ErrorModule : Array[0..31] of Bool;   // Module error
         PNSlaveWarning { ExternalAccessible := 'False'; ExternalVisible := 'False'; ExternalWritable := 'False'} : Bool;   // Profinet slave has a warning
      END_STRUCT;
   END_STRUCT;

END_TYPE

FUNCTION "FC_GetDevicePN" : Void
TITLE = FC_GetDevicePN
{ S7_Optimized_Access := 'TRUE' }
AUTHOR : MHSE
VERSION : 3.0
// ATTRIBUTES
// AUTO_NUMBER = True
// BLOCK_NUMBER = 18
// END_ATTRIBUTES
   VAR_INPUT
      is_PNDeviceName : String;   // Name of the device
      ix_SimulationModeActive : Bool;   // True = Simulation mode active
   END_VAR

   VAR_IN_OUT
      iqUDT_PND : "UDT_PNDevice";   // Device found in Profinet structure
   END_VAR

   VAR_TEMP
      ti_NrOfConfiguredPNNetworks : Int;   // Number of networks configured in project
      ti_NrOfDevices : Int;   // Nr of devices is networks
      ti_LcPNNetworkNumber : Int;   // Loop counter to find PN network number
      ti_LcPNDeviceNumber : Int;   // Loop counter to find PN device number
   END_VAR


BEGIN
	(*
	----------------------------------------------------------------------------------------

	Version history:
	Date        | Version   | Author        | Remark
	----------------------------------------------------------------------------------------
	16/09/2019  | 2.3       | F.Baten       | Cut out of 'FB_RIO'
	29/09/2019  | 2.4       | K.Pokorski    | Network seach started from 1 instead 0
	30/09/2019  | 2.5       | K.Pokorski    | Chagne prefixes of temporary varaibles from 'si' to 'ti'
	12/11/2019  | 3.0       | P.Majka       | 3.0 MHS library release TIA 15.1
	21/02/2023  | 4.0       | F.Baten       | 4.0 Release TIA 17.5
	*)

	REGION 1 - Get Device Profinet number
	    // if simulation is disabled
	    IF NOT #ix_SimulationModeActive
	    THEN
	        // And the profinet device is not found yet
	        IF (#is_PNDeviceName <> "DB_ProfinetDiagnostic".ProfinetNetworks[#iqUDT_PND.PNNetworknumber].DeviceStatus[#iqUDT_PND.PNDeviceNumber].DeviceState.PNDeviceName)
	            OR #iqUDT_PND.PNDeviceFound = FALSE
	        THEN
	            #iqUDT_PND.PNDeviceFound := FALSE;

	            // check how many profinet networks are configured
	            #ti_NrOfConfiguredPNNetworks := "FC_GetNrOfArrayEl"("DB_ProfinetDiagnostic".ProfinetNetworks);

	            FOR #ti_LcPNNetworkNumber := 1 TO (#ti_NrOfConfiguredPNNetworks) DO

	                #iqUDT_PND.PNNetworknumber := #ti_LcPNNetworkNumber;

	                // and check how many devices are configured per network
	                #ti_NrOfDevices := "FC_GetNrOfArrayEl"("DB_ProfinetDiagnostic".ProfinetNetworks[#iqUDT_PND.PNNetworknumber].DeviceStatus);

	                // check for each of the devices in the networks if the PN device name is similair to the configured device name
	                FOR #ti_LcPNDeviceNumber := 0 TO (#ti_NrOfDevices - 1) DO

	                    #iqUDT_PND.PNDeviceNumber := #ti_LcPNDeviceNumber;

	                    // set device found when a match is found for the device name in the PN network
	                    IF (#is_PNDeviceName = "DB_ProfinetDiagnostic".ProfinetNetworks[#iqUDT_PND.PNNetworknumber].DeviceStatus[#iqUDT_PND.PNDeviceNumber].DeviceState.PNDeviceName
	                        AND #is_PNDeviceName <> '')
	                    THEN

	                        #iqUDT_PND.PNDeviceFound := TRUE;
	                        EXIT;

	                    END_IF;
	                END_FOR;

	                // exit loop when device name is matching
	                IF #iqUDT_PND.PNDeviceFound
	                THEN

	                    EXIT;

	                END_IF;
	            END_FOR;
	        END_IF;
	    END_IF;

	END_REGION
END_FUNCTION

FUNCTION "FC_GetPNPortStatus" : Void
{ S7_Optimized_Access := 'TRUE' }
VERSION : 0.1
// ATTRIBUTES
// AUTO_NUMBER = True
// BLOCK_NUMBER = 20
// END_ATTRIBUTES
   VAR_INPUT
      ii_NumberOfPorts : Int;   //  Number of ports in device
      iUDT_DevicePNInfo : "UDT_PNDevice";   //  PN device info structure
   END_VAR

   VAR_OUTPUT
      qa_PortFault : Array[1..8] of Bool;   //  When TRUE then specific port has a fault
   END_VAR

   VAR_TEMP
      tp_GetDiagInfo {InstructionName := 'DIS'; LibVersion := '1.0'} : DIS;   //  Diagnostic structure
      tp_DeviceGeoAddr {InstructionName := 'GEOADDR'; LibVersion := '1.0'} : GEOADDR;   //  Device pointer structre
      ta_PortFault : Array[1..8] of Bool;   //  When TRUE then port has a fault
      ti_Geo2LogStatus : Int;   //  GEO2LOG status code
      ti_GetDiagStatus : Int;   //  Get_Diag status code
      ti_Log2GeoStatus : Int;   //  LOG2GEO status code
      ti_Loopcounter : Int;   //  Loop counter
      tui_cnt : UInt;   //  Not used
      tdi_PortLaddr : HW_ANY;   //  HW identifier
      ti_PortFault : Bool;   //  At least one port is faulty
      tx_ConfigurationError : Bool;   //  Configuration error occurred
   END_VAR

   VAR CONSTANT
      ci_Area : UInt := 1;   //     Area ID of IO Profinet devices
      ci_HWTYPE : UInt := 5;
      ci_PortSlot : UInt := 0;
      ci_PortSubslot : Word := 16#8000;
   END_VAR


BEGIN
	(*
	----------------------------------------------------------------------------------------

	Version history:
	Date        | Version   | Author        | Remark
	----------------------------------------------------------------------------------------
	03/11/2020  | 3.0       | K.Pokorski    | first release MHS TIA 15.1
	17/12/2020  | 3.1       | K.Pokorski    | Run operation only during error
	21/02/2023  | 4.0       | F.Baten       | 4.0 Release TIA 17.5
	*)

	REGION 1 - Check configuration

	    #tx_ConfigurationError := #ii_NumberOfPorts < 1
	    OR #ii_NumberOfPorts > 8
	    OR NOT #iUDT_DevicePNInfo.PNDeviceFound;

	END_REGION

	REGION 2 - Read profinet network number

	    // Using LOG2GEO profinet network address is read
	    #ti_Log2GeoStatus := LOG2GEO(LADDR := "DB_ProfinetDiagnostic".ProfinetNetworks[#iUDT_DevicePNInfo.PNNetworknumber].DeviceStatus[#iUDT_DevicePNInfo.PNDeviceNumber].DeviceState.HW_ID,
	                                 GEOADDR := #tp_DeviceGeoAddr);

	END_REGION

	REGION 3 - Preparation the device pointer

	    // HWTYPE = 5 - Submodule
	    #tp_DeviceGeoAddr.HWTYPE := #ci_HWTYPE;
	    // AREA = 1 - PROFINET IO
	    #tp_DeviceGeoAddr.AREA := #ci_Area;
	    // SLOT = 0 - Ports are on slot 0
	    #tp_DeviceGeoAddr.SLOT := #ci_PortSlot;
	    // STATION - Profinet number
	    #tp_DeviceGeoAddr.STATION := "DB_ProfinetDiagnostic".ProfinetNetworks[#iUDT_DevicePNInfo.PNNetworknumber].DeviceStatus[#iUDT_DevicePNInfo.PNDeviceNumber].DeviceState.ProfinetNumber;

	END_REGION

	REGION 4 - Checking the port status
	    // If device report error and is available on the PN network
	    IF "DB_ProfinetDiagnostic".ProfinetNetworks[#iUDT_DevicePNInfo.PNNetworknumber].DeviceStatus[#iUDT_DevicePNInfo.PNDeviceNumber].DeviceState.Error
	        AND "DB_ProfinetDiagnostic".ProfinetNetworks[#iUDT_DevicePNInfo.PNNetworknumber].DeviceStatus[#iUDT_DevicePNInfo.PNDeviceNumber].DeviceState.Exist
	        AND NOT #tx_ConfigurationError
	    THEN

	        // Loop through all profinet ports
	        FOR #ti_Loopcounter := 1 TO #ii_NumberOfPorts DO
	            // Reset auxiliary port fault bit
	            #ta_PortFault[#ti_Loopcounter] := FALSE;
	            // SUBSLOT = 16#8000 plus port number (TIA structure to refer to port)
	            #tp_DeviceGeoAddr.SUBSLOT := INT_TO_UINT(WORD_TO_INT(#ci_PortSubslot) + (#ti_Loopcounter));
	            // Using GEO2LOG port address is read
	            #ti_Geo2LogStatus := GEO2LOG(GEOADDR := #tp_DeviceGeoAddr, LADDR => #tdi_PortLaddr);
	            // Using GET_DIAG port status is read
	            #ti_GetDiagStatus := GET_DIAG(MODE := 1, LADDR := #tdi_PortLaddr, CNT_DIAG => #tui_cnt, DIAG := #tp_GetDiagInfo);

	            // Set port fault if all operations do not report any error and port is faulty
	            IF #ti_GetDiagStatus = 0
	                AND #ti_Geo2LogStatus = 0
	                AND #ti_Log2GeoStatus = 0
	                AND #tp_GetDiagInfo.OwnState = 4
	            THEN
	                #ta_PortFault[#ti_Loopcounter] := TRUE;
	            END_IF;
	        END_FOR;
	        // Reset module status if error occurred
	    ELSIF #tx_ConfigurationError
	    THEN
	        FOR #ti_Loopcounter := 1 TO 8 DO
	            #ta_PortFault[#ti_Loopcounter] := FALSE;
	        END_FOR;
	    END_IF;

	END_REGION

	REGION 5 - Write output

	    #qa_PortFault := #ta_PortFault;

	END_REGION


END_FUNCTION

